gfCNCPoint3[1224] = {X 357.0844, Y 26.7729, Z -3.8333, A 0.000, B 0.000, C 0.000 }
gfCNCPoint3[1225] = {X 357.1951, Y 25.0733, Z -3.8333, A 0.000, B 0.000, C 0.000 }
gfCNCPoint3[1226] = {X 357.1435, Y 23.3709, Z -3.8333, A 0.000, B 0.000, C 0.000 }
gfCNCPoint3[1227] = {X 356.9299, Y 21.6811, Z -3.8333, A 0.000, B 0.000, C 0.000 }
gfCNCPoint3[1228] = {X 356.5958, Y 20.2415, Z -3.8333, A 0.000, B 0.000, C 0.000 }
gfCNCPoint3[1229] = {X 356.0861, Y 18.8543, Z -3.8333, A 0.000, B 0.000, C 0.000 }
gfCNCPoint3[1230] = {X 355.4086, Y 17.5409, Z -3.8333, A 0.000, B 0.000, C 0.000 }
gfCNCPoint3[1231] = {X 354.5737, Y 16.3214, Z -3.8333, A 0.000, B 0.000, C 0.000 }
gfCNCPoint3[1232] = {X 353.6956, Y 15.3423, Z -3.8333, A 0.000, B 0.000, C 0.000 }
gfCNCPoint3[1233] = {X 352.6863, Y 14.4990, Z -3.8333, A 0.000, B 0.000, C 0.000 }
gfCNCPoint3[1234] = {X 351.5666, Y 13.8090, Z -3.8333, A 0.000, B 0.000, C 0.000 }
gfCNCPoint3[1235] = {X 350.3596, Y 13.2864, Z -3.8333, A 0.000, B 0.000, C 0.000 }
gfCNCPoint3[1236] = {X 349.0902, Y 12.9422, Z -3.8333, A 0.000, B 0.000, C 0.000 }
gfCNCPoint3[1237] = {X 347.3476, Y 12.7251, Z -3.8333, A 0.000, B 0.000, C 0.000 }
gfCNCPoint3[1238] = {X 345.5915, Y 12.7393, Z -3.8333, A 0.000, B 0.000, C 0.000 }
gfCNCPoint3[1239] = {X 343.8527, Y 12.9848, Z -3.8333, A 0.000, B 0.000, C 0.000 }
gfCNCPoint3[1240] = {X 342.1613, Y 13.4572, Z -3.8333, A 0.000, B 0.000, C 0.000 }
gfCNCPoint3[1241] = {X 340.5469, Y 14.1483, Z -3.8333, A 0.000, B 0.000, C 0.000 }
gfCNCPoint3[1242] = {X 339.0376, Y 15.0460, Z -3.8333, A 0.000, B 0.000, C 0.000 }
gfCNCPoint3[1243] = {X 338.9896, Y 15.9040, Z -3.8333, A 0.000, B 0.000, C 0.000 }
gfCNCPoint3[1244] = {X 338.7758, Y 16.7364, Z -3.8333, A 0.000, B 0.000, C 0.000 }
gfCNCPoint3[1245] = {X 338.4043, Y 17.5112, Z -3.8333, A 0.000, B 0.000, C 0.000 }
gfCNCPoint3[1246] = {X 337.8893, Y 18.1991, Z -3.8333, A 0.000, B 0.000, C 0.000 }
gfCNCPoint3[1247] = {X 337.2504, Y 18.7738, Z -3.8333, A 0.000, B 0.000, C 0.000 }
gfCNCPoint3[1248] = {X 336.5606, Y 19.2813, Z -3.8333, A 0.000, B 0.000, C 0.000 }
gfCNCPoint3[1249] = {X 335.7284, Y 19.7495, Z -3.8333, A 0.000, B 0.000, C 0.000 }
gfCNCPoint3[1250] = {X 334.8148, Y 20.0271, Z -3.8333, A 0.000, B 0.000, C 0.000 }
gfCNCPoint3[1251] = {X 333.8628, Y 20.1012, Z -3.8333, A 0.000, B 0.000, C 0.000 }
gfCNCPoint3[1252] = {X 332.9173, Y 19.9681, Z -3.8333, A 0.000, B 0.000, C 0.000 }
gfCNCPoint3[1253] = {X 332.0228, Y 19.6341, Z -3.8333, A 0.000, B 0.000, C 0.000 }
gfCNCPoint3[1254] = {X 331.2213, Y 19.1151, Z -3.8333, A 0.000, B 0.000, C 0.000 }
gfCNCPoint3[1255] = {X 330.5507, Y 18.4353, Z -3.8333, A 0.000, B 0.000, C 0.000 }
gfCNCPoint3[1256] = {X 330.0425, Y 17.6269, Z -3.8333, A 0.000, B 0.000, C 0.000 }
gfCNCPoint3[1257] = {X 326.5223, Y 10.3852, Z -3.8333, A 0.000, B 0.000, C 0.000 }
gfCNCPoint3[1258] = {X 326.2154, Y 9.5469, Z -3.8333, A 0.000, B 0.000, C 0.000 }
gfCNCPoint3[1259] = {X 326.0841, Y 8.6639, Z -3.8333, A 0.000, B 0.000, C 0.000 }
gfCNCPoint3[1260] = {X 326.1338, Y 7.7725, Z -3.8333, A 0.000, B 0.000, C 0.000 }
gfCNCPoint3[1261] = {X 326.3623, Y 6.9096, Z -3.8333, A 0.000, B 0.000, C 0.000 }
gfCNCPoint3[1262] = {X 326.7603, Y 6.1105, Z -3.8333, A 0.000, B 0.000, C 0.000 }
gfCNCPoint3[1263] = {X 327.3114, Y 5.4082, Z -3.8333, A 0.000, B 0.000, C 0.000 }
gfCNCPoint3[1264] = {X 327.9929, Y 4.8316, Z -3.8333, A 0.000, B 0.000, C 0.000 }
gfCNCPoint3[1265] = {X 328.6647, Y 4.3715, Z -3.8333, A 0.000, B 0.000, C 0.000 }
gfCNCPoint3[1266] = {X 329.5525, Y 3.9111, Z -3.8333, A 0.000, B 0.000, C 0.000 }
gfCNCPoint3[1267] = {X 330.5213, Y 3.6631, Z -3.8333, A 0.000, B 0.000, C 0.000 }
gfCNCPoint3[1268] = {X 331.5211, Y 3.6402, Z -3.8333, A 0.000, B 0.000, C 0.000 }
gfCNCPoint3[1269] = {X 332.5003, Y 3.8437, Z -3.8333, A 0.000, B 0.000, C 0.000 }
gfCNCPoint3[1270] = {X 333.5103, Y 3.2689, Z -3.8333, A 0.000, B 0.000, C 0.000 }
gfCNCPoint3[1271] = {X 334.5430, Y 2.7360, Z -3.8333, A 0.000, B 0.000, C 0.000 }
gfCNCPoint3[1272] = {X 334.3316, Y 2.3050, Z -3.8333, A 0.000, B 0.000, C 0.000 }
gfCNCPoint3[1273] = {X 2.3035, Y 2.3050, Z -3.8333, A 0.000, B 0.000, C 0.000 }
gfCNCPoint3[1274] = {X 2.3035, Y 6.8597, Z -3.8333, A 0.000, B 0.000, C 0.000 }
gfCNCPoint3[1275] = {X 2.4041, Y 6.8798, Z -3.8333, A 0.000, B 0.000, C 0.000 }
gfCNCPoint3[1276] = {X 2.8649, Y 6.6913, Z -3.8333, A 0.000, B 0.000, C 0.000 }
gfCNCPoint3[1277] = {X 3.3320, Y 6.5189, Z -3.8333, A 0.000, B 0.000, C 0.000 }
gfCNCPoint3[1278] = {X 5.4373, Y 5.7870, Z -3.8333, A 0.000, B 0.000, C 0.000 }
gfCNCPoint3[1279] = {X 7.5978, Y 5.2386, Z -3.8333, A 0.000, B 0.000, C 0.000 }
gfCNCPoint3[1280] = {X 9.7973, Y 4.8776, Z -3.8333, A 0.000, B 0.000, C 0.000 }
gfCNCPoint3[1281] = {X 12.0197, Y 4.7069, Z -3.8333, A 0.000, B 0.000, C 0.000 }
gfCNCPoint3[1282] = {X 14.2486, Y 4.7276, Z -3.8333, A 0.000, B 0.000, C 0.000 }
gfCNCPoint3[1283] = {X 16.4674, Y 4.9396, Z -3.8333, A 0.000, B 0.000, C 0.000 }
gfCNCPoint3[1284] = {X 18.0965, Y 5.2204, Z -3.8333, A 0.000, B 0.000, C 0.000 }
gfCNCPoint3[1285] = {X 19.6967, Y 5.6352, Z -3.8333, A 0.000, B 0.000, C 0.000 }
gfCNCPoint3[1286] = {X 21.2571, Y 6.1811, Z -3.8333, A 0.000, B 0.000, C 0.000 }
gfCNCPoint3[1287] = {X 22.7668, Y 6.8545, Z -3.8333, A 0.000, B 0.000, C 0.000 }
gfCNCPoint3[1288] = {X 24.4883, Y 7.8186, Z -3.8333, A 0.000, B 0.000, C 0.000 }
gfCNCPoint3[1289] = {X 26.1061, Y 8.9481, Z -3.8333, A 0.000, B 0.000, C 0.000 }
gfCNCPoint3[1290] = {X 27.4003, Y 10.0783, Z -3.8333, A 0.000, B 0.000, C 0.000 }
gfCNCPoint3[1291] = {X 28.5612, Y 11.3450, Z -3.8333, A 0.000, B 0.000, C 0.000 }
gfCNCPoint3[1292] = {X 29.5745, Y 12.7325, Z -3.8333, A 0.000, B 0.000, C 0.000 }
gfCNCPoint3[1293] = {X 30.4278, Y 14.2239, Z -3.8333, A 0.000, B 0.000, C 0.000 }
gfCNCPoint3[1294] = {X 31.1104, Y 15.8006, Z -3.8333, A 0.000, B 0.000, C 0.000 }
gfCNCPoint3[1295] = {X 31.6697, Y 17.7362, Z -3.8333, A 0.000, B 0.000, C 0.000 }
gfCNCPoint3[1296] = {X 32.0027, Y 19.7232, Z -3.8333, A 0.000, B 0.000, C 0.000 }
gfCNCPoint3[1297] = {X 32.1050, Y 21.7354, Z -3.8333, A 0.000, B 0.000, C 0.000 }
gfCNCPoint3[1298] = {X 31.9753, Y 23.7459, Z -3.8333, A 0.000, B 0.000, C 0.000 }
gfCNCPoint3[1299] = {X 31.6152, Y 25.7282, Z -3.8333, A 0.000, B 0.000, C 0.000 }
gfCNCPoint3[1300] = {X 31.1690, Y 27.2346, Z -3.8333, A 0.000, B 0.000, C 0.000 }
gfCNCPoint3[1301] = {X 30.5588, Y 28.6823, Z -3.8333, A 0.000, B 0.000, C 0.000 }
gfCNCPoint3[1302] = {X 29.7921, Y 30.0536, Z -3.8333, A 0.000, B 0.000, C 0.000 }
gfCNCPoint3[1303] = {X 29.4475, Y 30.5712, Z -3.8333, A 0.000, B 0.000, C 0.000 }
gfCNCPoint3[1304] = {X 29.0806, Y 31.0733, Z -3.8333, A 0.000, B 0.000, C 0.000 }
gfCNCPoint3[1305] = {X 29.6385, Y 31.7919, Z -3.8333, A 0.000, B 0.000, C 0.000 }
gfCNCPoint3[1306] = {X 30.0955, Y 32.5786, Z -3.8333, A 0.000, B 0.000, C 0.000 }
gfCNCPoint3[1307] = {X 33.1423, Y 38.8726, Z -3.8333, A 0.000, B 0.000, C 0.000 }
gfCNCPoint3[1308] = {X 33.5391, Y 39.8957, Z -3.8333, A 0.000, B 0.000, C 0.000 }
gfCNCPoint3[1309] = {X 33.7662, Y 40.9694, Z -3.8333, A 0.000, B 0.000, C 0.000 }
gfCNCPoint3[1310] = {X 33.8177, Y 42.0656, Z -3.8333, A 0.000, B 0.000, C 0.000 }
gfCNCPoint3[1311] = {X 33.7164, Y 43.0266, Z -3.8333, A 0.000, B 0.000, C 0.000 }
gfCNCPoint3[1312] = {X 33.4799, Y 43.9636, Z -3.8333, A 0.000, B 0.000, C 0.000 }
gfCNCPoint3[1313] = {X 33.1103, Y 44.8630, Z -3.8333, A 0.000, B 0.000, C 0.000 }
gfCNCPoint3[1314] = {X 32.6161, Y 45.7005, Z -3.8333, A 0.000, B 0.000, C 0.000 }
gfCNCPoint3[1315] = {X 32.0075, Y 46.4590, Z -3.8333, A 0.000, B 0.000, C 0.000 }
gfCNCPoint3[1316] = {X 31.2970, Y 47.1229, Z -3.8333, A 0.000, B 0.000, C 0.000 }
gfCNCPoint3[1317] = {X 30.7593, Y 47.5577, Z -3.8333, A 0.000, B 0.000, C 0.000 }
gfCNCPoint3[1318] = {X 29.8533, Y 48.1757, Z -3.8333, A 0.000, B 0.000, C 0.000 }
gfCNCPoint3[1319] = {X 28.8600, Y 48.6403, Z -3.8333, A 0.000, B 0.000, C 0.000 }
gfCNCPoint3[1320] = {X 27.8050, Y 48.9396, Z -3.8333, A 0.000, B 0.000, C 0.000 }
gfCNCPoint3[1321] = {X 26.7156, Y 49.0659, Z -3.8333, A 0.000, B 0.000, C 0.000 }
gfCNCPoint3[1322] = {X 25.6202, Y 49.0158, Z -3.8333, A 0.000, B 0.000, C 0.000 }
gfCNCPoint3[1323] = {X 23.9315, Y 49.8548, Z -3.8333, A 0.000, B 0.000, C 0.000 }
gfCNCPoint3[1324] = {X 22.1957, Y 50.5913, Z -3.8333, A 0.000, B 0.000, C 0.000 }
gfCNCPoint3[1325] = {X 20.4190, Y 51.2227, Z -3.8333, A 0.000, B 0.000, C 0.000 }
gfCNCPoint3[1326] = {X 18.3991, Y 51.7971, Z -3.8333, A 0.000, B 0.000, C 0.000 }
gfCNCPoint3[1327] = {X 16.3386, Y 52.2022, Z -3.8333, A 0.000, B 0.000, C 0.000 }
gfCNCPoint3[1328] = {X 14.2517, Y 52.4352, Z -3.8333, A 0.000, B 0.000, C 0.000 }
gfCNCPoint3[1329] = {X 12.1526, Y 52.4947, Z -3.8333, A 0.000, B 0.000, C 0.000 }
gfCNCPoint3[1330] = {X 10.0558, Y 52.3800, Z -3.8333, A 0.000, B 0.000, C 0.000 }
gfCNCPoint3[1331] = {X 7.9757, Y 52.0921, Z -3.8333, A 0.000, B 0.000, C 0.000 }
gfCNCPoint3[1332] = {X 6.6905, Y 51.8245, Z -3.8333, A 0.000, B 0.000, C 0.000 }
gfCNCPoint3[1333] = {X 5.4261, Y 51.4714, Z -3.8333, A 0.000, B 0.000, C 0.000 }
gfCNCPoint3[1334] = {X 3.8369, Y 50.8930, Z -3.8333, A 0.000, B 0.000, C 0.000 }
gfCNCPoint3[1335] = {X 2.3035, Y 50.1795, Z -3.8333, A 0.000, B 0.000, C 0.000 }
gfCNCPoint3[1336] = {X 2.3035, Y 97.6950, Z -3.8333, A 0.000, B 0.000, C 0.000 }
gfCNCPoint3[1337] = {X 120.1200, Y 97.6950, Z -3.8333, A 0.000, B 0.000, C 0.000 }
gfCNCPoint3[1338] = {X 120.1200, Y 97.0659, Z -3.8333, A 0.000, B 0.000, C 0.000 }
gfCNCPoint3[1339] = {X 120.2339, Y 96.0179, Z -3.8333, A 0.000, B 0.000, C 0.000 }
gfCNCPoint3[1340] = {X 120.5702, Y 95.0187, Z -3.8333, A 0.000, B 0.000, C 0.000 }
gfCNCPoint3[1341] = {X 121.1132, Y 94.1151, Z -3.8333, A 0.000, B 0.000, C 0.000 }
gfCNCPoint3[1342] = {X 121.8376, Y 93.3492, Z -3.8333, A 0.000, B 0.000, C 0.000 }
gfCNCPoint3[1343] = {X 122.7096, Y 92.7568, Z -3.8333, A 0.000, B 0.000, C 0.000 }
gfCNCPoint3[1344] = {X 123.6885, Y 92.3655, Z -3.8333, A 0.000, B 0.000, C 0.000 }
gfCNCPoint3[1345] = {X 124.7286, Y 92.1935, Z -3.8333, A 0.000, B 0.000, C 0.000 }
gfCNCPoint3[1346] = {X 124.7867, Y 92.1787, Z -3.8333, A 0.000, B 0.000, C 0.000 }
gfCNCPoint3[1347] = {X 124.8457, Y 92.1679, Z -3.8333, A 0.000, B 0.000, C 0.000 }
gfCNCPoint3[1348] = {X 125.3649, Y 92.0908, Z -3.8333, A 0.000, B 0.000, C 0.000 }
gfCNCPoint3[1349] = {X 126.0998, Y 91.9697, Z -3.8333, A 0.000, B 0.000, C 0.000 }
gfCNCPoint3[1350] = {X 126.8256, Y 91.8023, Z -3.8333, A 0.000, B 0.000, C 0.000 }
gfCNCPoint3[1351] = {X 127.9736, Y 90.7130, Z -3.8333, A 0.000, B 0.000, C 0.000 }
gfCNCPoint3[1352] = {X 129.0632, Y 89.5654, Z -3.8333, A 0.000, B 0.000, C 0.000 }
gfCNCPoint3[1353] = {X 154.9462, Y 61.1423, Z -3.8333, A 0.000, B 0.000, C 0.000 }
gfCNCPoint3[1354] = {X 154.6593, Y 60.4497, Z -3.8333, A 0.000, B 0.000, C 0.000 }
gfCNCPoint3[1355] = {X 154.4819, Y 59.7213, Z -3.8333, A 0.000, B 0.000, C 0.000 }
gfCNCPoint3[1356] = {X 154.4181, Y 58.9744, Z -3.8333, A 0.000, B 0.000, C 0.000 }
gfCNCPoint3[1357] = {X 154.4180, Y 58.0000, Z -3.8333, A 0.000, B 0.000, C 0.000 }
gfCNCPoint3[1358] = {X 154.5117, Y 57.0480, Z -3.8333, A 0.000, B 0.000, C 0.000 }
gfCNCPoint3[1359] = {X 154.7894, Y 56.1325, Z -3.8333, A 0.000, B 0.000, C 0.000 }
gfCNCPoint3[1360] = {X 155.2404, Y 55.2888, Z -3.8333, A 0.000, B 0.000, C 0.000 }
gfCNCPoint3[1361] = {X 155.8473, Y 54.5493, Z -3.8333, A 0.000, B 0.000, C 0.000 }
gfCNCPoint3[1362] = {X 156.5868, Y 53.9424, Z -3.8333, A 0.000, B 0.000, C 0.000 }
gfCNCPoint3[1363] = {X 157.4305, Y 53.4915, Z -3.8333, A 0.000, B 0.000, C 0.000 }
gfCNCPoint3[1364] = {X 158.3459, Y 53.2138, Z -3.8333, A 0.000, B 0.000, C 0.000 }
gfCNCPoint3[1365] = {X 159.2980, Y 53.1200, Z -3.8333, A 0.000, B 0.000, C 0.000 }
gfCNCPoint3[1366] = {X 178.5335, Y 53.1200, Z -3.8333, A 0.000, B 0.000, C 0.000 }
gfCNCPoint3[1367] = {X 179.4855, Y 53.2138, Z -3.8333, A 0.000, B 0.000, C 0.000 }
gfCNCPoint3[1368] = {X 180.4010, Y 53.4915, Z -3.8333, A 0.000, B 0.000, C 0.000 }
gfCNCPoint3[1369] = {X 181.2447, Y 53.9424, Z -3.8333, A 0.000, B 0.000, C 0.000 }
gfCNCPoint3[1370] = {X 181.9842, Y 54.5493, Z -3.8333, A 0.000, B 0.000, C 0.000 }
gfCNCPoint3[1371] = {X 182.5911, Y 55.2888, Z -3.8333, A 0.000, B 0.000, C 0.000 }
gfCNCPoint3[1372] = {X 183.0420, Y 56.1325, Z -3.8333, A 0.000, B 0.000, C 0.000 }
gfCNCPoint3[1373] = {X 183.3197, Y 57.0480, Z -3.8333, A 0.000, B 0.000, C 0.000 }
gfCNCPoint3[1374] = {X 183.4135, Y 58.0000, Z -3.8333, A 0.000, B 0.000, C 0.000 }
gfCNCPoint3[1375] = {X 183.4133, Y 58.9744, Z -3.8333, A 0.000, B 0.000, C 0.000 }
gfCNCPoint3[1376] = {X 183.3512, Y 59.7113, Z -3.8333, A 0.000, B 0.000, C 0.000 }
gfCNCPoint3[1377] = {X 183.1784, Y 60.4304, Z -3.8333, A 0.000, B 0.000, C 0.000 }
gfCNCPoint3[1378] = {X 182.8990, Y 61.1152, Z -3.8333, A 0.000, B 0.000, C 0.000 }
gfCNCPoint3[1379] = {X 209.8913, Y 90.5758, Z -3.8333, A 0.000, B 0.000, C 0.000 }
gfCNCPoint3[1380] = {X 210.5201, Y 91.2137, Z -3.8333, A 0.000, B 0.000, C 0.000 }
gfCNCPoint3[1381] = {X 211.1937, Y 91.8042, Z -3.8333, A 0.000, B 0.000, C 0.000 }
gfCNCPoint3[1382] = {X 211.3597, Y 91.9086, Z -3.8333, A 0.000, B 0.000, C 0.000 }
gfCNCPoint3[1383] = {X 211.5461, Y 91.9696, Z -3.8333, A 0.000, B 0.000, C 0.000 }
gfCNCPoint3[1384] = {X 212.2018, Y 92.1098, Z -3.8333, A 0.000, B 0.000, C 0.000 }
gfCNCPoint3[1385] = {X 213.4083, Y 92.2618, Z -3.8333, A 0.000, B 0.000, C 0.000 }
gfCNCPoint3[1386] = {X 214.4425, Y 92.1756, Z -3.8333, A 0.000, B 0.000, C 0.000 }
gfCNCPoint3[1387] = {X 215.4785, Y 92.1166, Z -3.8333, A 0.000, B 0.000, C 0.000 }
gfCNCPoint3[1388] = {X 216.0525, Y 92.0568, Z -3.8333, A 0.000, B 0.000, C 0.000 }
gfCNCPoint3[1389] = {X 216.6054, Y 91.8915, Z -3.8333, A 0.000, B 0.000, C 0.000 }
gfCNCPoint3[1390] = {X 217.1180, Y 91.6265, Z -3.8333, A 0.000, B 0.000, C 0.000 }
gfCNCPoint3[1391] = {X 244.6013, Y 74.0195, Z -3.8333, A 0.000, B 0.000, C 0.000 }
gfCNCPoint3[1392] = {X 221.4278, Y 64.9254, Z -3.8333, A 0.000, B 0.000, C 0.000 }
gfCNCPoint3[1393] = {X 219.7200, Y 64.3531, Z -3.8333, A 0.000, B 0.000, C 0.000 }
gfCNCPoint3[1394] = {X 217.9579, Y 63.9800, Z -3.8333, A 0.000, B 0.000, C 0.000 }
gfCNCPoint3[1395] = {X 216.1647, Y 63.8112, Z -3.8333, A 0.000, B 0.000, C 0.000 }
gfCNCPoint3[1396] = {X 215.1121, Y 63.6594, Z -3.8333, A 0.000, B 0.000, C 0.000 }
gfCNCPoint3[1397] = {X 214.1174, Y 63.2832, Z -3.8333, A 0.000, B 0.000, C 0.000 }
gfCNCPoint3[1398] = {X 213.2278, Y 62.7005, Z -3.8333, A 0.000, B 0.000, C 0.000 }
gfCNCPoint3[1399] = {X 212.4856, Y 61.9389, Z -3.8333, A 0.000, B 0.000, C 0.000 }
gfCNCPoint3[1400] = {X 211.9260, Y 61.0346, Z -3.8333, A 0.000, B 0.000, C 0.000 }
gfCNCPoint3[1401] = {X 211.5756, Y 60.0305, Z -3.8333, A 0.000, B 0.000, C 0.000 }
gfCNCPoint3[1402] = {X 211.4510, Y 58.9744, Z -3.8333, A 0.000, B 0.000, C 0.000 }
gfCNCPoint3[1403] = {X 211.4508, Y 58.0000, Z -3.8333, A 0.000, B 0.000, C 0.000 }
gfCNCPoint3[1404] = {X 211.5446, Y 57.0480, Z -3.8333, A 0.000, B 0.000, C 0.000 }
gfCNCPoint3[1405] = {X 211.8223, Y 56.1325, Z -3.8333, A 0.000, B 0.000, C 0.000 }
gfCNCPoint3[1406] = {X 212.2732, Y 55.2888, Z -3.8333, A 0.000, B 0.000, C 0.000 }
gfCNCPoint3[1407] = {X 212.8801, Y 54.5493, Z -3.8333, A 0.000, B 0.000, C 0.000 }
gfCNCPoint3[1408] = {X 213.6196, Y 53.9424, Z -3.8333, A 0.000, B 0.000, C 0.000 }
gfCNCPoint3[1409] = {X 214.4633, Y 53.4915, Z -3.8333, A 0.000, B 0.000, C 0.000 }
gfCNCPoint3[1410] = {X 215.3788, Y 53.2138, Z -3.8333, A 0.000, B 0.000, C 0.000 }
gfCNCPoint3[1411] = {X 216.3308, Y 53.1200, Z -3.8333, A 0.000, B 0.000, C 0.000 }
gfCNCPoint3[1412] = {X 237.2617, Y 53.1200, Z -3.8333, A 0.000, B 0.000, C 0.000 }
gfCNCPoint3[1413] = {X 238.3265, Y 53.2376, Z -3.8333, A 0.000, B 0.000, C 0.000 }
gfCNCPoint3[1414] = {X 239.3400, Y 53.5847, Z -3.8333, A 0.000, B 0.000, C 0.000 }
gfCNCPoint3[1415] = {X 240.2534, Y 54.1446, Z -3.8333, A 0.000, B 0.000, C 0.000 }
gfCNCPoint3[1416] = {X 241.0226, Y 54.8903, Z -3.8333, A 0.000, B 0.000, C 0.000 }
gfCNCPoint3[1417] = {X 241.6105, Y 55.7859, Z -3.8333, A 0.000, B 0.000, C 0.000 }
gfCNCPoint3[1418] = {X 241.9888, Y 56.7881, Z -3.8333, A 0.000, B 0.000, C 0.000 }
gfCNCPoint3[1419] = {X 242.1393, Y 57.8488, Z -3.8333, A 0.000, B 0.000, C 0.000 }
gfCNCPoint3[1420] = {X 247.6958, Y 60.0148, Z -3.8333, A 0.000, B 0.000, C 0.000 }
gfCNCPoint3[1421] = {X 275.0731, Y 70.8777, Z -3.8333, A 0.000, B 0.000, C 0.000 }
gfCNCPoint3[1422] = {X 275.0726, Y 63.6742, Z -3.8333, A 0.000, B 0.000, C 0.000 }
gfCNCPoint3[1423] = {X 274.0643, Y 63.3058, Z -3.8333, A 0.000, B 0.000, C 0.000 }
gfCNCPoint3[1424] = {X 273.1609, Y 62.7260, Z -3.8333, A 0.000, B 0.000, C 0.000 }
gfCNCPoint3[1425] = {X 272.4062, Y 61.9626, Z -3.8333, A 0.000, B 0.000, C 0.000 }
gfCNCPoint3[1426] = {X 271.8366, Y 61.0527, Z -3.8333, A 0.000, B 0.000, C 0.000 }
gfCNCPoint3[1427] = {X 271.4797, Y 60.0403, Z -3.8333, A 0.000, B 0.000, C 0.000 }
gfCNCPoint3[1428] = {X 271.3529, Y 58.9744, Z -3.8333, A 0.000, B 0.000, C 0.000 }
gfCNCPoint3[1429] = {X 271.3527, Y 58.0000, Z -3.8333, A 0.000, B 0.000, C 0.000 }
gfCNCPoint3[1430] = {X 271.4465, Y 57.0480, Z -3.8333, A 0.000, B 0.000, C 0.000 }
gfCNCPoint3[1431] = {X 271.7242, Y 56.1325, Z -3.8333, A 0.000, B 0.000, C 0.000 }
gfCNCPoint3[1432] = {X 272.1751, Y 55.2888, Z -3.8333, A 0.000, B 0.000, C 0.000 }
gfCNCPoint3[1433] = {X 272.7820, Y 54.5493, Z -3.8333, A 0.000, B 0.000, C 0.000 }
gfCNCPoint3[1434] = {X 273.5215, Y 53.9424, Z -3.8333, A 0.000, B 0.000, C 0.000 }
gfCNCPoint3[1435] = {X 274.3652, Y 53.4915, Z -3.8333, A 0.000, B 0.000, C 0.000 }
gfCNCPoint3[1436] = {X 275.2806, Y 53.2138, Z -3.8333, A 0.000, B 0.000, C 0.000 }
gfCNCPoint3[1437] = {X 276.2327, Y 53.1200, Z -3.8333, A 0.000, B 0.000, C 0.000 }
gfCNCPoint3[1438] = {X 292.7731, Y 53.1200, Z -3.8333, A 0.000, B 0.000, C 0.000 }
gfCNCPoint3[1439] = {X 293.7251, Y 53.2138, Z -3.8333, A 0.000, B 0.000, C 0.000 }
gfCNCPoint3[1440] = {X 294.6406, Y 53.4915, Z -3.8333, A 0.000, B 0.000, C 0.000 }
gfCNCPoint3[1441] = {X 295.4843, Y 53.9424, Z -3.8333, A 0.000, B 0.000, C 0.000 }
gfCNCPoint3[1442] = {X 296.2238, Y 54.5493, Z -3.8333, A 0.000, B 0.000, C 0.000 }
gfCNCPoint3[1443] = {X 296.8307, Y 55.2888, Z -3.8333, A 0.000, B 0.000, C 0.000 }
gfCNCPoint3[1444] = {X 297.2816, Y 56.1325, Z -3.8333, A 0.000, B 0.000, C 0.000 }
gfCNCPoint3[1445] = {X 297.5593, Y 57.0480, Z -3.8333, A 0.000, B 0.000, C 0.000 }
gfCNCPoint3[1446] = {X 297.6531, Y 58.0000, Z -3.8333, A 0.000, B 0.000, C 0.000 }
gfCNCPoint3[1447] = {X 297.6531, Y 58.9370, Z -3.8333, A 0.000, B 0.000, C 0.000 }
gfCNCPoint3[1448] = {X 297.5307, Y 60.0092, Z -3.8333, A 0.000, B 0.000, C 0.000 }
gfCNCPoint3[1449] = {X 297.1764, Y 61.0286, Z -3.8333, A 0.000, B 0.000, C 0.000 }
gfCNCPoint3[1450] = {X 296.6074, Y 61.9456, Z -3.8333, A 0.000, B 0.000, C 0.000 }
gfCNCPoint3[1451] = {X 295.8514, Y 62.7156, Z -3.8333, A 0.000, B 0.000, C 0.000 }
gfCNCPoint3[1452] = {X 294.9451, Y 63.3014, Z -3.8333, A 0.000, B 0.000, C 0.000 }
gfCNCPoint3[1453] = {X 293.9324, Y 63.6745, Z -3.8333, A 0.000, B 0.000, C 0.000 }
gfCNCPoint3[1454] = {X 293.9324, Y 92.3204, Z -3.8333, A 0.000, B 0.000, C 0.000 }
gfCNCPoint3[1455] = {X 294.9449, Y 92.6960, Z -3.8333, A 0.000, B 0.000, C 0.000 }
gfCNCPoint3[1456] = {X 295.8509, Y 93.2837, Z -3.8333, A 0.000, B 0.000, C 0.000 }
gfCNCPoint3[1457] = {X 296.6066, Y 94.0552, Z -3.8333, A 0.000, B 0.000, C 0.000 }
gfCNCPoint3[1458] = {X 297.1754, Y 94.9731, Z -3.8333, A 0.000, B 0.000, C 0.000 }
gfCNCPoint3[1459] = {X 297.5300, Y 95.9932, Z -3.8333, A 0.000, B 0.000, C 0.000 }
gfCNCPoint3[1460] = {X 297.6531, Y 97.0661, Z -3.8333, A 0.000, B 0.000, C 0.000 }
gfCNCPoint3[1461] = {X 297.6531, Y 97.6950, Z -3.8333, A 0.000, B 0.000, C 0.000 }
gfCNCPoint3[1462] = {X 297.1731, Y 97.6950, Z -3.8333, A 0.000, B 0.000, C 0.000 }
gfCNCPoint3[1463] = {X 297.1731, Y 98.0000, Z -3.8333, A 0.000, B 0.000, C 0.000 }
gfCNCPoint3[1464] = {X 297.0628, Y 98.9791, Z -3.8333, A 0.000, B 0.000, C 0.000 }
gfCNCPoint3[1465] = {X 296.7373, Y 99.9091, Z -3.8333, A 0.000, B 0.000, C 0.000 }
gfCNCPoint3[1466] = {X 296.2131, Y 100.7434, Z -3.8333, A 0.000, B 0.000, C 0.000 }
gfCNCPoint3[1467] = {X 295.5164, Y 101.4401, Z -3.8333, A 0.000, B 0.000, C 0.000 }
gfCNCPoint3[1468] = {X 294.6822, Y 101.9643, Z -3.8333, A 0.000, B 0.000, C 0.000 }
gfCNCPoint3[1469] = {X 293.7522, Y 102.2897, Z -3.8333, A 0.000, B 0.000, C 0.000 }
gfCNCPoint3[1470] = {X 292.7731, Y 102.4000, Z -3.8333, A 0.000, B 0.000, C 0.000 }
gfCNCPoint3[1471] = {X 276.2327, Y 102.4000, Z -3.8333, A 0.000, B 0.000, C 0.000 }
gfCNCPoint3[1472] = {X 275.2536, Y 102.2897, Z -3.8333, A 0.000, B 0.000, C 0.000 }
gfCNCPoint3[1473] = {X 274.3236, Y 101.9643, Z -3.8333, A 0.000, B 0.000, C 0.000 }
gfCNCPoint3[1474] = {X 273.4893, Y 101.4401, Z -3.8333, A 0.000, B 0.000, C 0.000 }
gfCNCPoint3[1475] = {X 272.7926, Y 100.7434, Z -3.8333, A 0.000, B 0.000, C 0.000 }
gfCNCPoint3[1476] = {X 272.2684, Y 99.9091, Z -3.8333, A 0.000, B 0.000, C 0.000 }
gfCNCPoint3[1477] = {X 271.9430, Y 98.9791, Z -3.8333, A 0.000, B 0.000, C 0.000 }
gfCNCPoint3[1478] = {X 271.8327, Y 98.0000, Z -3.8333, A 0.000, B 0.000, C 0.000 }
gfCNCPoint3[1479] = {X 271.8329, Y 97.0190, Z -3.8333, A 0.000, B 0.000, C 0.000 }
gfCNCPoint3[1480] = {X 271.9305, Y 96.1432, Z -3.8333, A 0.000, B 0.000, C 0.000 }
gfCNCPoint3[1481] = {X 272.2006, Y 95.3045, Z -3.8333, A 0.000, B 0.000, C 0.000 }
gfCNCPoint3[1482] = {X 272.6325, Y 94.5364, Z -3.8333, A 0.000, B 0.000, C 0.000 }
gfCNCPoint3[1483] = {X 273.2087, Y 93.8698, Z -3.8333, A 0.000, B 0.000, C 0.000 }
gfCNCPoint3[1484] = {X 273.9062, Y 93.3313, Z -3.8333, A 0.000, B 0.000, C 0.000 }
gfCNCPoint3[1485] = {X 274.6970, Y 92.9426, Z -3.8333, A 0.000, B 0.000, C 0.000 }
gfCNCPoint3[1486] = {X 275.5494, Y 92.7193, Z -3.8333, A 0.000, B 0.000, C 0.000 }
gfCNCPoint3[1487] = {X 275.5494, Y 85.6495, Z -3.8333, A 0.000, B 0.000, C 0.000 }
gfCNCPoint3[1488] = {X 262.6481, Y 80.5922, Z -3.8333, A 0.000, B 0.000, C 0.000 }
gfCNCPoint3[1489] = {X 262.3197, Y 80.7991, Z -3.8333, A 0.000, B 0.000, C 0.000 }
gfCNCPoint3[1490] = {X 237.8767, Y 96.6314, Z -3.8333, A 0.000, B 0.000, C 0.000 }
gfCNCPoint3[1491] = {X 237.8798, Y 97.0659, Z -3.8333, A 0.000, B 0.000, C 0.000 }
gfCNCPoint3[1492] = {X 237.8798, Y 98.0000, Z -3.8333, A 0.000, B 0.000, C 0.000 }
gfCNCPoint3[1493] = {X 237.7695, Y 98.9791, Z -3.8333, A 0.000, B 0.000, C 0.000 }
gfCNCPoint3[1494] = {X 237.4440, Y 99.9091, Z -3.8333, A 0.000, B 0.000, C 0.000 }
gfCNCPoint3[1495] = {X 236.9198, Y 100.7434, Z -3.8333, A 0.000, B 0.000, C 0.000 }
gfCNCPoint3[1496] = {X 236.2231, Y 101.4401, Z -3.8333, A 0.000, B 0.000, C 0.000 }
gfCNCPoint3[1497] = {X 235.3889, Y 101.9643, Z -3.8333, A 0.000, B 0.000, C 0.000 }
gfCNCPoint3[1498] = {X 234.4589, Y 102.2897, Z -3.8333, A 0.000, B 0.000, C 0.000 }
gfCNCPoint3[1499] = {X 233.4798, Y 102.4000, Z -3.8333, A 0.000, B 0.000, C 0.000 }
gfCNCPoint3[1500] = {X 214.1790, Y 102.4000, Z -3.8333, A 0.000, B 0.000, C 0.000 }
gfCNCPoint3[1501] = {X 213.7862, Y 102.3824, Z -3.8333, A 0.000, B 0.000, C 0.000 }
gfCNCPoint3[1502] = {X 213.3966, Y 102.3299, Z -3.8333, A 0.000, B 0.000, C 0.000 }
gfCNCPoint3[1503] = {X 213.0069, Y 102.3824, Z -3.8333, A 0.000, B 0.000, C 0.000 }
gfCNCPoint3[1504] = {X 212.6141, Y 102.4000, Z -3.8333, A 0.000, B 0.000, C 0.000 }
gfCNCPoint3[1505] = {X 194.9870, Y 102.4000, Z -3.8333, A 0.000, B 0.000, C 0.000 }
gfCNCPoint3[1506] = {X 194.0079, Y 102.2897, Z -3.8333, A 0.000, B 0.000, C 0.000 }
gfCNCPoint3[1507] = {X 193.0779, Y 101.9643, Z -3.8333, A 0.000, B 0.000, C 0.000 }
gfCNCPoint3[1508] = {X 192.2436, Y 101.4401, Z -3.8333, A 0.000, B 0.000, C 0.000 }
gfCNCPoint3[1509] = {X 191.5469, Y 100.7434, Z -3.8333, A 0.000, B 0.000, C 0.000 }
gfCNCPoint3[1510] = {X 191.0227, Y 99.9091, Z -3.8333, A 0.000, B 0.000, C 0.000 }
gfCNCPoint3[1511] = {X 190.6973, Y 98.9791, Z -3.8333, A 0.000, B 0.000, C 0.000 }
gfCNCPoint3[1512] = {X 190.5870, Y 98.0000, Z -3.8333, A 0.000, B 0.000, C 0.000 }
gfCNCPoint3[1513] = {X 190.5870, Y 97.0659, Z -3.8333, A 0.000, B 0.000, C 0.000 }
gfCNCPoint3[1514] = {X 190.6897, Y 96.1207, Z -3.8333, A 0.000, B 0.000, C 0.000 }
gfCNCPoint3[1515] = {X 190.9931, Y 95.2196, Z -3.8333, A 0.000, B 0.000, C 0.000 }
gfCNCPoint3[1516] = {X 191.4830, Y 94.4047, Z -3.8333, A 0.000, B 0.000, C 0.000 }
gfCNCPoint3[1517] = {X 188.5295, Y 91.1802, Z -3.8333, A 0.000, B 0.000, C 0.000 }
gfCNCPoint3[1518] = {X 150.1254, Y 91.1802, Z -3.8333, A 0.000, B 0.000, C 0.000 }
gfCNCPoint3[1519] = {X 147.2494, Y 94.3664, Z -3.8333, A 0.000, B 0.000, C 0.000 }
gfCNCPoint3[1520] = {X 147.7554, Y 95.1907, Z -3.8333, A 0.000, B 0.000, C 0.000 }
gfCNCPoint3[1521] = {X 148.0703, Y 96.1051, Z -3.8333, A 0.000, B 0.000, C 0.000 }
gfCNCPoint3[1522] = {X 148.1791, Y 97.0661, Z -3.8333, A 0.000, B 0.000, C 0.000 }
gfCNCPoint3[1523] = {X 148.1791, Y 98.0000, Z -3.8333, A 0.000, B 0.000, C 0.000 }
gfCNCPoint3[1524] = {X 148.0688, Y 98.9791, Z -3.8333, A 0.000, B 0.000, C 0.000 }
gfCNCPoint3[1525] = {X 147.7434, Y 99.9091, Z -3.8333, A 0.000, B 0.000, C 0.000 }
gfCNCPoint3[1526] = {X 147.2192, Y 100.7434, Z -3.8333, A 0.000, B 0.000, C 0.000 }
gfCNCPoint3[1527] = {X 146.5225, Y 101.4401, Z -3.8333, A 0.000, B 0.000, C 0.000 }
gfCNCPoint3[1528] = {X 145.6882, Y 101.9643, Z -3.8333, A 0.000, B 0.000, C 0.000 }
gfCNCPoint3[1529] = {X 144.7582, Y 102.2897, Z -3.8333, A 0.000, B 0.000, C 0.000 }
gfCNCPoint3[1530] = {X 143.7791, Y 102.4000, Z -3.8333, A 0.000, B 0.000, C 0.000 }
gfCNCPoint3[1531] = {X 125.0000, Y 102.4000, Z -3.8333, A 0.000, B 0.000, C 0.000 }
gfCNCPoint3[1532] = {X 124.0209, Y 102.2897, Z -3.8333, A 0.000, B 0.000, C 0.000 }
gfCNCPoint3[1533] = {X 123.0909, Y 101.9643, Z -3.8333, A 0.000, B 0.000, C 0.000 }
gfCNCPoint3[1534] = {X 122.2566, Y 101.4401, Z -3.8333, A 0.000, B 0.000, C 0.000 }
gfCNCPoint3[1535] = {X 121.5599, Y 100.7434, Z -3.8333, A 0.000, B 0.000, C 0.000 }
gfCNCPoint3[1536] = {X 121.0357, Y 99.9091, Z -3.8333, A 0.000, B 0.000, C 0.000 }
gfCNCPoint3[1537] = {X 120.7103, Y 98.9791, Z -3.8333, A 0.000, B 0.000, C 0.000 }
gfCNCPoint3[1538] = {X 120.6000, Y 98.0000, Z -3.8333, A 0.000, B 0.000, C 0.000 }
gfCNCPoint3[1539] = {X 120.6000, Y 97.0659, Z -3.8333, A 0.000, B 0.000, C 0.000 }
gfCNCPoint3[1540] = {X 120.7047, Y 96.1120, Z -3.8333, A 0.000, B 0.000, C 0.000 }
gfCNCPoint3[1541] = {X 121.0137, Y 95.2034, Z -3.8333, A 0.000, B 0.000, C 0.000 }
gfCNCPoint3[1542] = {X 121.5123, Y 94.3834, Z -3.8333, A 0.000, B 0.000, C 0.000 }
gfCNCPoint3[1543] = {X 122.1769, Y 93.6910, Z -3.8333, A 0.000, B 0.000, C 0.000 }
gfCNCPoint3[1544] = {X 122.9757, Y 93.1592, Z -3.8333, A 0.000, B 0.000, C 0.000 }
gfCNCPoint3[1545] = {X 123.8709, Y 92.8133, Z -3.8333, A 0.000, B 0.000, C 0.000 }
gfCNCPoint3[1546] = {X 124.8198, Y 92.6696, Z -3.8333, A 0.000, B 0.000, C 0.000 }
gfCNCPoint3[1547] = {X 124.8671, Y 92.6531, Z -3.8333, A 0.000, B 0.000, C 0.000 }
gfCNCPoint3[1548] = {X 124.9162, Y 92.6427, Z -3.8333, A 0.000, B 0.000, C 0.000 }
gfCNCPoint3[1549] = {X 125.4412, Y 92.5648, Z -3.8333, A 0.000, B 0.000, C 0.000 }
gfCNCPoint3[1550] = {X 126.2566, Y 92.4278, Z -3.8333, A 0.000, B 0.000, C 0.000 }
gfCNCPoint3[1551] = {X 127.0610, Y 92.2360, Z -3.8333, A 0.000, B 0.000, C 0.000 }
gfCNCPoint3[1552] = {X 128.2728, Y 91.0926, Z -3.8333, A 0.000, B 0.000, C 0.000 }
gfCNCPoint3[1553] = {X 129.4210, Y 89.8854, Z -3.8333, A 0.000, B 0.000, C 0.000 }
gfCNCPoint3[1554] = {X 133.5081, Y 85.3895, Z -3.8333, A 0.000, B 0.000, C 0.000 }
gfCNCPoint3[1555] = {X 155.5329, Y 61.2109, Z -3.8333, A 0.000, B 0.000, C 0.000 }
gfCNCPoint3[1556] = {X 155.1840, Y 60.4948, Z -3.8333, A 0.000, B 0.000, C 0.000 }
gfCNCPoint3[1557] = {X 154.9701, Y 59.7274, Z -3.8333, A 0.000, B 0.000, C 0.000 }
gfCNCPoint3[1558] = {X 154.8980, Y 58.9340, Z -3.8333, A 0.000, B 0.000, C 0.000 }
gfCNCPoint3[1559] = {X 154.8980, Y 58.0000, Z -3.8333, A 0.000, B 0.000, C 0.000 }
gfCNCPoint3[1560] = {X 155.0083, Y 57.0209, Z -3.8333, A 0.000, B 0.000, C 0.000 }
gfCNCPoint3[1561] = {X 155.3337, Y 56.0909, Z -3.8333, A 0.000, B 0.000, C 0.000 }
gfCNCPoint3[1562] = {X 155.8579, Y 55.2566, Z -3.8333, A 0.000, B 0.000, C 0.000 }
gfCNCPoint3[1563] = {X 156.5546, Y 54.5599, Z -3.8333, A 0.000, B 0.000, C 0.000 }
gfCNCPoint3[1564] = {X 157.3889, Y 54.0357, Z -3.8333, A 0.000, B 0.000, C 0.000 }
gfCNCPoint3[1565] = {X 158.3189, Y 53.7103, Z -3.8333, A 0.000, B 0.000, C 0.000 }
gfCNCPoint3[1566] = {X 159.2980, Y 53.6000, Z -3.8333, A 0.000, B 0.000, C 0.000 }
gfCNCPoint3[1567] = {X 178.5335, Y 53.6000, Z -3.8333, A 0.000, B 0.000, C 0.000 }
gfCNCPoint3[1568] = {X 179.5126, Y 53.7103, Z -3.8333, A 0.000, B 0.000, C 0.000 }
gfCNCPoint3[1569] = {X 180.4426, Y 54.0357, Z -3.8333, A 0.000, B 0.000, C 0.000 }
gfCNCPoint3[1570] = {X 181.2769, Y 54.5599, Z -3.8333, A 0.000, B 0.000, C 0.000 }
gfCNCPoint3[1571] = {X 181.9736, Y 55.2566, Z -3.8333, A 0.000, B 0.000, C 0.000 }
gfCNCPoint3[1572] = {X 182.4978, Y 56.0909, Z -3.8333, A 0.000, B 0.000, C 0.000 }
gfCNCPoint3[1573] = {X 182.8232, Y 57.0209, Z -3.8333, A 0.000, B 0.000, C 0.000 }
gfCNCPoint3[1574] = {X 182.9335, Y 58.0000, Z -3.8333, A 0.000, B 0.000, C 0.000 }
gfCNCPoint3[1575] = {X 182.9334, Y 58.9704, Z -3.8333, A 0.000, B 0.000, C 0.000 }
gfCNCPoint3[1576] = {X 182.8587, Y 59.7419, Z -3.8333, A 0.000, B 0.000, C 0.000 }
gfCNCPoint3[1577] = {X 182.6499, Y 60.4883, Z -3.8333, A 0.000, B 0.000, C 0.000 }
gfCNCPoint3[1578] = {X 182.3133, Y 61.1865, Z -3.8333, A 0.000, B 0.000, C 0.000 }
gfCNCPoint3[1579] = {X 209.5374, Y 90.9000, Z -3.8333, A 0.000, B 0.000, C 0.000 }
gfCNCPoint3[1580] = {X 210.1907, Y 91.5629, Z -3.8333, A 0.000, B 0.000, C 0.000 }
gfCNCPoint3[1581] = {X 210.8906, Y 92.1765, Z -3.8333, A 0.000, B 0.000, C 0.000 }
gfCNCPoint3[1582] = {X 211.1522, Y 92.3414, Z -3.8333, A 0.000, B 0.000, C 0.000 }
gfCNCPoint3[1583] = {X 211.4457, Y 92.4390, Z -3.8333, A 0.000, B 0.000, C 0.000 }
gfCNCPoint3[1584] = {X 212.1215, Y 92.5835, Z -3.8333, A 0.000, B 0.000, C 0.000 }
gfCNCPoint3[1585] = {X 213.4015, Y 92.7447, Z -3.8333, A 0.000, B 0.000, C 0.000 }
gfCNCPoint3[1586] = {X 214.4547, Y 92.6560, Z -3.8333, A 0.000, B 0.000, C 0.000 }
gfCNCPoint3[1587] = {X 215.5099, Y 92.5958, Z -3.8333, A 0.000, B 0.000, C 0.000 }
gfCNCPoint3[1588] = {X 216.1640, Y 92.5237, Z -3.8333, A 0.000, B 0.000, C 0.000 }
gfCNCPoint3[1589] = {X 216.7937, Y 92.3330, Z -3.8333, A 0.000, B 0.000, C 0.000 }
gfCNCPoint3[1590] = {X 217.3778, Y 92.0300, Z -3.8333, A 0.000, B 0.000, C 0.000 }
gfCNCPoint3[1591] = {X 222.9188, Y 88.4542, Z -3.8333, A 0.000, B 0.000, C 0.000 }
gfCNCPoint3[1592] = {X 245.6531, Y 73.9167, Z -3.8333, A 0.000, B 0.000, C 0.000 }
gfCNCPoint3[1593] = {X 221.6008, Y 64.4777, Z -3.8333, A 0.000, B 0.000, C 0.000 }
gfCNCPoint3[1594] = {X 219.8423, Y 63.8889, Z -3.8333, A 0.000, B 0.000, C 0.000 }
gfCNCPoint3[1595] = {X 218.0279, Y 63.5052, Z -3.8333, A 0.000, B 0.000, C 0.000 }
gfCNCPoint3[1596] = {X 216.1816, Y 63.3315, Z -3.8333, A 0.000, B 0.000, C 0.000 }
gfCNCPoint3[1597] = {X 215.2274, Y 63.1935, Z -3.8333, A 0.000, B 0.000, C 0.000 }
gfCNCPoint3[1598] = {X 214.3262, Y 62.8509, Z -3.8333, A 0.000, B 0.000, C 0.000 }
gfCNCPoint3[1599] = {X 213.5213, Y 62.3203, Z -3.8333, A 0.000, B 0.000, C 0.000 }
gfCNCPoint3[1600] = {X 212.8512, Y 61.6271, Z -3.8333, A 0.000, B 0.000, C 0.000 }
gfCNCPoint3[1601] = {X 212.3482, Y 60.8046, Z -3.8333, A 0.000, B 0.000, C 0.000 }
gfCNCPoint3[1602] = {X 212.0364, Y 59.8923, Z -3.8333, A 0.000, B 0.000, C 0.000 }
gfCNCPoint3[1603] = {X 211.9308, Y 58.9340, Z -3.8333, A 0.000, B 0.000, C 0.000 }
gfCNCPoint3[1604] = {X 211.9308, Y 58.0000, Z -3.8333, A 0.000, B 0.000, C 0.000 }
gfCNCPoint3[1605] = {X 212.0411, Y 57.0209, Z -3.8333, A 0.000, B 0.000, C 0.000 }
gfCNCPoint3[1606] = {X 212.3665, Y 56.0909, Z -3.8333, A 0.000, B 0.000, C 0.000 }
gfCNCPoint3[1607] = {X 212.8907, Y 55.2566, Z -3.8333, A 0.000, B 0.000, C 0.000 }
gfCNCPoint3[1608] = {X 213.5875, Y 54.5599, Z -3.8333, A 0.000, B 0.000, C 0.000 }
gfCNCPoint3[1609] = {X 214.4217, Y 54.0357, Z -3.8333, A 0.000, B 0.000, C 0.000 }
gfCNCPoint3[1610] = {X 215.3517, Y 53.7103, Z -3.8333, A 0.000, B 0.000, C 0.000 }
gfCNCPoint3[1611] = {X 216.3308, Y 53.6000, Z -3.8333, A 0.000, B 0.000, C 0.000 }
gfCNCPoint3[1612] = {X 237.2617, Y 53.6000, Z -3.8333, A 0.000, B 0.000, C 0.000 }
gfCNCPoint3[1613] = {X 238.2408, Y 53.7103, Z -3.8333, A 0.000, B 0.000, C 0.000 }
gfCNCPoint3[1614] = {X 239.1708, Y 54.0357, Z -3.8333, A 0.000, B 0.000, C 0.000 }
gfCNCPoint3[1615] = {X 240.0050, Y 54.5599, Z -3.8333, A 0.000, B 0.000, C 0.000 }
gfCNCPoint3[1616] = {X 240.7017, Y 55.2566, Z -3.8333, A 0.000, B 0.000, C 0.000 }
gfCNCPoint3[1617] = {X 241.2260, Y 56.0909, Z -3.8333, A 0.000, B 0.000, C 0.000 }
gfCNCPoint3[1618] = {X 241.5514, Y 57.0209, Z -3.8333, A 0.000, B 0.000, C 0.000 }
gfCNCPoint3[1619] = {X 241.6617, Y 58.0000, Z -3.8333, A 0.000, B 0.000, C 0.000 }
gfCNCPoint3[1620] = {X 241.6617, Y 58.1778, Z -3.8333, A 0.000, B 0.000, C 0.000 }
gfCNCPoint3[1621] = {X 247.5187, Y 60.4610, Z -3.8333, A 0.000, B 0.000, C 0.000 }
gfCNCPoint3[1622] = {X 275.5531, Y 71.5846, Z -3.8333, A 0.000, B 0.000, C 0.000 }
gfCNCPoint3[1623] = {X 275.5525, Y 63.2812, Z -3.8333, A 0.000, B 0.000, C 0.000 }
gfCNCPoint3[1624] = {X 274.6933, Y 63.0560, Z -3.8333, A 0.000, B 0.000, C 0.000 }
gfCNCPoint3[1625] = {X 273.8967, Y 62.6628, Z -3.8333, A 0.000, B 0.000, C 0.000 }
gfCNCPoint3[1626] = {X 273.1954, Y 62.1176, Z -3.8333, A 0.000, B 0.000, C 0.000 }
gfCNCPoint3[1627] = {X 272.6179, Y 61.4427, Z -3.8333, A 0.000, B 0.000, C 0.000 }
gfCNCPoint3[1628] = {X 272.1877, Y 60.6655, Z -3.8333, A 0.000, B 0.000, C 0.000 }
gfCNCPoint3[1629] = {X 271.9224, Y 59.8178, Z -3.8333, A 0.000, B 0.000, C 0.000 }
gfCNCPoint3[1630] = {X 271.8327, Y 58.9340, Z -3.8333, A 0.000, B 0.000, C 0.000 }
gfCNCPoint3[1631] = {X 271.8327, Y 58.0000, Z -3.8333, A 0.000, B 0.000, C 0.000 }
gfCNCPoint3[1632] = {X 271.9430, Y 57.0209, Z -3.8333, A 0.000, B 0.000, C 0.000 }
gfCNCPoint3[1633] = {X 272.2684, Y 56.0909, Z -3.8333, A 0.000, B 0.000, C 0.000 }
gfCNCPoint3[1634] = {X 272.7926, Y 55.2566, Z -3.8333, A 0.000, B 0.000, C 0.000 }
gfCNCPoint3[1635] = {X 273.4893, Y 54.5599, Z -3.8333, A 0.000, B 0.000, C 0.000 }
gfCNCPoint3[1636] = {X 274.3236, Y 54.0357, Z -3.8333, A 0.000, B 0.000, C 0.000 }
gfCNCPoint3[1637] = {X 275.2536, Y 53.7103, Z -3.8333, A 0.000, B 0.000, C 0.000 }
gfCNCPoint3[1638] = {X 276.2327, Y 53.6000, Z -3.8333, A 0.000, B 0.000, C 0.000 }
gfCNCPoint3[1639] = {X 292.7731, Y 53.6000, Z -3.8333, A 0.000, B 0.000, C 0.000 }
gfCNCPoint3[1640] = {X 293.7522, Y 53.7103, Z -3.8333, A 0.000, B 0.000, C 0.000 }
gfCNCPoint3[1641] = {X 294.6822, Y 54.0357, Z -3.8333, A 0.000, B 0.000, C 0.000 }
gfCNCPoint3[1642] = {X 295.5164, Y 54.5599, Z -3.8333, A 0.000, B 0.000, C 0.000 }
gfCNCPoint3[1643] = {X 296.2131, Y 55.2566, Z -3.8333, A 0.000, B 0.000, C 0.000 }
gfCNCPoint3[1644] = {X 296.7373, Y 56.0909, Z -3.8333, A 0.000, B 0.000, C 0.000 }
gfCNCPoint3[1645] = {X 297.0628, Y 57.0209, Z -3.8333, A 0.000, B 0.000, C 0.000 }
gfCNCPoint3[1646] = {X 297.1731, Y 58.0000, Z -3.8333, A 0.000, B 0.000, C 0.000 }
gfCNCPoint3[1647] = {X 297.1731, Y 58.9354, Z -3.8333, A 0.000, B 0.000, C 0.000 }
gfCNCPoint3[1648] = {X 297.0810, Y 59.8183, Z -3.8333, A 0.000, B 0.000, C 0.000 }
gfCNCPoint3[1649] = {X 296.8143, Y 60.6650, Z -3.8333, A 0.000, B 0.000, C 0.000 }
gfCNCPoint3[1650] = {X 296.3836, Y 61.4412, Z -3.8333, A 0.000, B 0.000, C 0.000 }
gfCNCPoint3[1651] = {X 295.8063, Y 62.1157, Z -3.8333, A 0.000, B 0.000, C 0.000 }
gfCNCPoint3[1652] = {X 295.1059, Y 62.6610, Z -3.8333, A 0.000, B 0.000, C 0.000 }
gfCNCPoint3[1653] = {X 294.3106, Y 63.0553, Z -3.8333, A 0.000, B 0.000, C 0.000 }
gfCNCPoint3[1654] = {X 293.4524, Y 63.2826, Z -3.8333, A 0.000, B 0.000, C 0.000 }
gfCNCPoint3[1655] = {X 293.4524, Y 92.7111, Z -3.8333, A 0.000, B 0.000, C 0.000 }
gfCNCPoint3[1656] = {X 294.3104, Y 92.9409, Z -3.8333, A 0.000, B 0.000, C 0.000 }
gfCNCPoint3[1657] = {X 295.1052, Y 93.3371, Z -3.8333, A 0.000, B 0.000, C 0.000 }
gfCNCPoint3[1658] = {X 295.8052, Y 93.8838, Z -3.8333, A 0.000, B 0.000, C 0.000 }
gfCNCPoint3[1659] = {X 296.3821, Y 94.5591, Z -3.8333, A 0.000, B 0.000, C 0.000 }
gfCNCPoint3[1660] = {X 296.8128, Y 95.3358, Z -3.8333, A 0.000, B 0.000, C 0.000 }
gfCNCPoint3[1661] = {X 297.0801, Y 96.1828, Z -3.8333, A 0.000, B 0.000, C 0.000 }
gfCNCPoint3[1662] = {X 297.1731, Y 97.0661, Z -3.8333, A 0.000, B 0.000, C 0.000 }
gfCNCPoint3[1663] = {X 297.1731, Y 97.6950, Z -3.8333, A 0.000, B 0.000, C 0.000 }
gfCNCPoint3[1664] = {X 297.6531, Y 97.6950, Z -3.8333, A 0.000, B 0.000, C 0.000 }
gfCNCPoint3[1665] = {X 314.2152, Y 97.6950, Z -3.8333, A 0.000, B 0.000, C 0.000 }
gfCNCPoint3[1666] = {X 313.0165, Y 96.8444, Z -3.8333, A 0.000, B 0.000, C 0.000 }
gfCNCPoint3[1667] = {X 311.8817, Y 95.9102, Z -3.8333, A 0.000, B 0.000, C 0.000 }
gfCNCPoint3[1668] = {X 310.9060, Y 94.9484, Z -3.8333, A 0.000, B 0.000, C 0.000 }
gfCNCPoint3[1669] = {X 310.0417, Y 93.8854, Z -3.8333, A 0.000, B 0.000, C 0.000 }
gfCNCPoint3[1670] = {X 309.2077, Y 92.5708, Z -3.8333, A 0.000, B 0.000, C 0.000 }
gfCNCPoint3[1671] = {X 308.5440, Y 91.1625, Z -3.8333, A 0.000, B 0.000, C 0.000 }
gfCNCPoint3[1672] = {X 308.0608, Y 89.6825, Z -3.8333, A 0.000, B 0.000, C 0.000 }
gfCNCPoint3[1673] = {X 307.7074, Y 88.0127, Z -3.8333, A 0.000, B 0.000, C 0.000 }
gfCNCPoint3[1674] = {X 307.4985, Y 86.3187, Z -3.8333, A 0.000, B 0.000, C 0.000 }
gfCNCPoint3[1675] = {X 307.4357, Y 84.6130, Z -3.8333, A 0.000, B 0.000, C 0.000 }
gfCNCPoint3[1676] = {X 307.4369, Y 63.6744, Z -3.8333, A 0.000, B 0.000, C 0.000 }
gfCNCPoint3[1677] = {X 306.4284, Y 63.3062, Z -3.8333, A 0.000, B 0.000, C 0.000 }
gfCNCPoint3[1678] = {X 305.5249, Y 62.7263, Z -3.8333, A 0.000, B 0.000, C 0.000 }
gfCNCPoint3[1679] = {X 304.7700, Y 61.9630, Z -3.8333, A 0.000, B 0.000, C 0.000 }
gfCNCPoint3[1680] = {X 304.2002, Y 61.0530, Z -3.8333, A 0.000, B 0.000, C 0.000 }
gfCNCPoint3[1681] = {X 303.8433, Y 60.0404, Z -3.8333, A 0.000, B 0.000, C 0.000 }
gfCNCPoint3[1682] = {X 303.7164, Y 58.9744, Z -3.8333, A 0.000, B 0.000, C 0.000 }
gfCNCPoint3[1683] = {X 303.7162, Y 58.0000, Z -3.8333, A 0.000, B 0.000, C 0.000 }
gfCNCPoint3[1684] = {X 303.8100, Y 57.0480, Z -3.8333, A 0.000, B 0.000, C 0.000 }
gfCNCPoint3[1685] = {X 304.0877, Y 56.1325, Z -3.8333, A 0.000, B 0.000, C 0.000 }
gfCNCPoint3[1686] = {X 304.5387, Y 55.2888, Z -3.8333, A 0.000, B 0.000, C 0.000 }
gfCNCPoint3[1687] = {X 305.1455, Y 54.5493, Z -3.8333, A 0.000, B 0.000, C 0.000 }
gfCNCPoint3[1688] = {X 305.8850, Y 53.9424, Z -3.8333, A 0.000, B 0.000, C 0.000 }
gfCNCPoint3[1689] = {X 306.7287, Y 53.4915, Z -3.8333, A 0.000, B 0.000, C 0.000 }
gfCNCPoint3[1690] = {X 307.6442, Y 53.2138, Z -3.8333, A 0.000, B 0.000, C 0.000 }
gfCNCPoint3[1691] = {X 308.5962, Y 53.1200, Z -3.8333, A 0.000, B 0.000, C 0.000 }
gfCNCPoint3[1692] = {X 324.3107, Y 53.1200, Z -3.8333, A 0.000, B 0.000, C 0.000 }
gfCNCPoint3[1693] = {X 325.2627, Y 53.2138, Z -3.8333, A 0.000, B 0.000, C 0.000 }
gfCNCPoint3[1694] = {X 326.1782, Y 53.4915, Z -3.8333, A 0.000, B 0.000, C 0.000 }
gfCNCPoint3[1695] = {X 327.0219, Y 53.9424, Z -3.8333, A 0.000, B 0.000, C 0.000 }
gfCNCPoint3[1696] = {X 327.7614, Y 54.5493, Z -3.8333, A 0.000, B 0.000, C 0.000 }
gfCNCPoint3[1697] = {X 328.3683, Y 55.2888, Z -3.8333, A 0.000, B 0.000, C 0.000 }
gfCNCPoint3[1698] = {X 328.8192, Y 56.1325, Z -3.8333, A 0.000, B 0.000, C 0.000 }
gfCNCPoint3[1699] = {X 329.0969, Y 57.0480, Z -3.8333, A 0.000, B 0.000, C 0.000 }
gfCNCPoint3[1700] = {X 329.1907, Y 58.0000, Z -3.8333, A 0.000, B 0.000, C 0.000 }
gfCNCPoint3[1701] = {X 329.1907, Y 58.9341, Z -3.8333, A 0.000, B 0.000, C 0.000 }
gfCNCPoint3[1702] = {X 329.0670, Y 60.0067, Z -3.8333, A 0.000, B 0.000, C 0.000 }
gfCNCPoint3[1703] = {X 328.7123, Y 61.0264, Z -3.8333, A 0.000, B 0.000, C 0.000 }
gfCNCPoint3[1704] = {X 328.1437, Y 61.9442, Z -3.8333, A 0.000, B 0.000, C 0.000 }
gfCNCPoint3[1705] = {X 327.3885, Y 62.7159, Z -3.8333, A 0.000, B 0.000, C 0.000 }
gfCNCPoint3[1706] = {X 326.4832, Y 63.3042, Z -3.8333, A 0.000, B 0.000, C 0.000 }
gfCNCPoint3[1707] = {X 325.4713, Y 63.6808, Z -3.8333, A 0.000, B 0.000, C 0.000 }
gfCNCPoint3[1708] = {X 325.4729, Y 83.2269, Z -3.8333, A 0.000, B 0.000, C 0.000 }
gfCNCPoint3[1709] = {X 325.4864, Y 84.6073, Z -3.8333, A 0.000, B 0.000, C 0.000 }
gfCNCPoint3[1710] = {X 325.5523, Y 85.7201, Z -3.8333, A 0.000, B 0.000, C 0.000 }
gfCNCPoint3[1711] = {X 325.7425, Y 86.8185, Z -3.8333, A 0.000, B 0.000, C 0.000 }
gfCNCPoint3[1712] = {X 325.8865, Y 86.9527, Z -3.8333, A 0.000, B 0.000, C 0.000 }
gfCNCPoint3[1713] = {X 326.0548, Y 87.0548, Z -3.8333, A 0.000, B 0.000, C 0.000 }
gfCNCPoint3[1714] = {X 326.4834, Y 87.2970, Z -3.8333, A 0.000, B 0.000, C 0.000 }
gfCNCPoint3[1715] = {X 327.8568, Y 87.8654, Z -3.8333, A 0.000, B 0.000, C 0.000 }
gfCNCPoint3[1716] = {X 329.2840, Y 88.2810, Z -3.8333, A 0.000, B 0.000, C 0.000 }
gfCNCPoint3[1717] = {X 332.3217, Y 88.8893, Z -3.8333, A 0.000, B 0.000, C 0.000 }
gfCNCPoint3[1718] = {X 335.3954, Y 89.2773, Z -3.8333, A 0.000, B 0.000, C 0.000 }
gfCNCPoint3[1719] = {X 339.5149, Y 89.5962, Z -3.8333, A 0.000, B 0.000, C 0.000 }
gfCNCPoint3[1720] = {X 343.6430, Y 89.7751, Z -3.8333, A 0.000, B 0.000, C 0.000 }
gfCNCPoint3[1721] = {X 347.7747, Y 89.8137, Z -3.8333, A 0.000, B 0.000, C 0.000 }
gfCNCPoint3[1722] = {X 352.1398, Y 89.7758, Z -3.8333, A 0.000, B 0.000, C 0.000 }
gfCNCPoint3[1723] = {X 356.5008, Y 89.5808, Z -3.8333, A 0.000, B 0.000, C 0.000 }
gfCNCPoint3[1724] = {X 360.8519, Y 89.2291, Z -3.8333, A 0.000, B 0.000, C 0.000 }
gfCNCPoint3[1725] = {X 363.1336, Y 88.9455, Z -3.8333, A 0.000, B 0.000, C 0.000 }
gfCNCPoint3[1726] = {X 365.3941, Y 88.5252, Z -3.8333, A 0.000, B 0.000, C 0.000 }
gfCNCPoint3[1727] = {X 367.6253, Y 87.9697, Z -3.8333, A 0.000, B 0.000, C 0.000 }
gfCNCPoint3[1728] = {X 368.9187, Y 87.4948, Z -3.8333, A 0.000, B 0.000, C 0.000 }
gfCNCPoint3[1729] = {X 370.1143, Y 86.8098, Z -3.8333, A 0.000, B 0.000, C 0.000 }
gfCNCPoint3[1730] = {X 370.2988, Y 85.3241, Z -3.8333, A 0.000, B 0.000, C 0.000 }
gfCNCPoint3[1731] = {X 370.3604, Y 83.8282, Z -3.8333, A 0.000, B 0.000, C 0.000 }
gfCNCPoint3[1732] = {X 370.3589, Y 63.6741, Z -3.8333, A 0.000, B 0.000, C 0.000 }
gfCNCPoint3[1733] = {X 369.3507, Y 63.3057, Z -3.8333, A 0.000, B 0.000, C 0.000 }
gfCNCPoint3[1734] = {X 368.4474, Y 62.7259, Z -3.8333, A 0.000, B 0.000, C 0.000 }
gfCNCPoint3[1735] = {X 367.6927, Y 61.9625, Z -3.8333, A 0.000, B 0.000, C 0.000 }
gfCNCPoint3[1736] = {X 367.1231, Y 61.0526, Z -3.8333, A 0.000, B 0.000, C 0.000 }
gfCNCPoint3[1737] = {X 366.7663, Y 60.0403, Z -3.8333, A 0.000, B 0.000, C 0.000 }
gfCNCPoint3[1738] = {X 366.6394, Y 58.9744, Z -3.8333, A 0.000, B 0.000, C 0.000 }
gfCNCPoint3[1739] = {X 366.6393, Y 58.0000, Z -3.8333, A 0.000, B 0.000, C 0.000 }
gfCNCPoint3[1740] = {X 366.7331, Y 57.0480, Z -3.8333, A 0.000, B 0.000, C 0.000 }
gfCNCPoint3[1741] = {X 367.0108, Y 56.1325, Z -3.8333, A 0.000, B 0.000, C 0.000 }
gfCNCPoint3[1742] = {X 367.4617, Y 55.2888, Z -3.8333, A 0.000, B 0.000, C 0.000 }
gfCNCPoint3[1743] = {X 368.0686, Y 54.5493, Z -3.8333, A 0.000, B 0.000, C 0.000 }
gfCNCPoint3[1744] = {X 368.8081, Y 53.9424, Z -3.8333, A 0.000, B 0.000, C 0.000 }
gfCNCPoint3[1745] = {X 369.6518, Y 53.4915, Z -3.8333, A 0.000, B 0.000, C 0.000 }
gfCNCPoint3[1746] = {X 370.5672, Y 53.2138, Z -3.8333, A 0.000, B 0.000, C 0.000 }
gfCNCPoint3[1747] = {X 371.5193, Y 53.1200, Z -3.8333, A 0.000, B 0.000, C 0.000 }
gfCNCPoint3[1748] = {X 388.0597, Y 53.1200, Z -3.8333, A 0.000, B 0.000, C 0.000 }
gfCNCPoint3[1749] = {X 389.0355, Y 53.2186, Z -3.8333, A 0.000, B 0.000, C 0.000 }
gfCNCPoint3[1750] = {X 389.9719, Y 53.5102, Z -3.8333, A 0.000, B 0.000, C 0.000 }
gfCNCPoint3[1751] = {X 390.8310, Y 53.9833, Z -3.8333, A 0.000, B 0.000, C 0.000 }
gfCNCPoint3[1752] = {X 391.5783, Y 54.6186, Z -3.8333, A 0.000, B 0.000, C 0.000 }
gfCNCPoint3[1753] = {X 392.1572, Y 55.3496, Z -3.8333, A 0.000, B 0.000, C 0.000 }
gfCNCPoint3[1754] = {X 392.5865, Y 56.1774, Z -3.8333, A 0.000, B 0.000, C 0.000 }
gfCNCPoint3[1755] = {X 392.8506, Y 57.0718, Z -3.8333, A 0.000, B 0.000, C 0.000 }
gfCNCPoint3[1756] = {X 392.9397, Y 58.0000, Z -3.8333, A 0.000, B 0.000, C 0.000 }
gfCNCPoint3[1757] = {X 392.9395, Y 58.9743, Z -3.8333, A 0.000, B 0.000, C 0.000 }
gfCNCPoint3[1758] = {X 392.8779, Y 59.7081, Z -3.8333, A 0.000, B 0.000, C 0.000 }
gfCNCPoint3[1759] = {X 392.7066, Y 60.4243, Z -3.8333, A 0.000, B 0.000, C 0.000 }
gfCNCPoint3[1760] = {X 392.4294, Y 61.1066, Z -3.8333, A 0.000, B 0.000, C 0.000 }
gfCNCPoint3[1761] = {X 392.0494, Y 61.7445, Z -3.8333, A 0.000, B 0.000, C 0.000 }
gfCNCPoint3[1762] = {X 391.5775, Y 62.3177, Z -3.8333, A 0.000, B 0.000, C 0.000 }
gfCNCPoint3[1763] = {X 390.8818, Y 62.9185, Z -3.8333, A 0.000, B 0.000, C 0.000 }
gfCNCPoint3[1764] = {X 390.0862, Y 63.3787, Z -3.8333, A 0.000, B 0.000, C 0.000 }
gfCNCPoint3[1765] = {X 389.2186, Y 63.6824, Z -3.8333, A 0.000, B 0.000, C 0.000 }
gfCNCPoint3[1766] = {X 389.2177, Y 73.4812, Z -3.8333, A 0.000, B 0.000, C 0.000 }
gfCNCPoint3[1767] = {X 398.8177, Y 73.4821, Z -3.8333, A 0.000, B 0.000, C 0.000 }
gfCNCPoint3[1768] = {X 398.8170, Y 80.5583, Z -3.8333, A 0.000, B 0.000, C 0.000 }
gfCNCPoint3[1769] = {X 405.8042, Y 76.0834, Z -3.8333, A 0.000, B 0.000, C 0.000 }
gfCNCPoint3[1770] = {X 400.0367, Y 73.8205, Z -3.8333, A 0.000, B 0.000, C 0.000 }
gfCNCPoint3[1771] = {X 399.4360, Y 73.6196, Z -3.8333, A 0.000, B 0.000, C 0.000 }
gfCNCPoint3[1772] = {X 398.8177, Y 73.4821, Z -3.8333, A 0.000, B 0.000, C 0.000 }
gfCNCPoint3[1773] = {X 396.4177, Y 73.4819, Z -3.8333, A 0.000, B 0.000, C 0.000 }
gfCNCPoint3[1774] = {X 396.4166, Y 84.5897, Z -3.8333, A 0.000, B 0.000, C 0.000 }
gfCNCPoint3[1775] = {X 396.4165, Y 84.9457, Z -3.8333, A 0.000, B 0.000, C 0.000 }
gfCNCPoint3[1776] = {X 411.0600, Y 75.5674, Z -3.8333, A 0.000, B 0.000, C 0.000 }
gfCNCPoint3[1777] = {X 400.9153, Y 71.5871, Z -3.8333, A 0.000, B 0.000, C 0.000 }
gfCNCPoint3[1778] = {X 399.6205, Y 71.1936, Z -3.8333, A 0.000, B 0.000, C 0.000 }
gfCNCPoint3[1779] = {X 398.2797, Y 71.0109, Z -3.8333, A 0.000, B 0.000, C 0.000 }
gfCNCPoint3[1780] = {X 397.3452, Y 70.9531, Z -3.8333, A 0.000, B 0.000, C 0.000 }
gfCNCPoint3[1781] = {X 396.4179, Y 70.8230, Z -3.8333, A 0.000, B 0.000, C 0.000 }
gfCNCPoint3[1782] = {X 396.4177, Y 73.4819, Z -3.8333, A 0.000, B 0.000, C 0.000 }
gfCNCPoint3[1783] = {X 394.0177, Y 73.4817, Z -3.8333, A 0.000, B 0.000, C 0.000 }
gfCNCPoint3[1784] = {X 394.0166, Y 84.5974, Z -3.8333, A 0.000, B 0.000, C 0.000 }
gfCNCPoint3[1785] = {X 394.0171, Y 84.7631, Z -3.8333, A 0.000, B 0.000, C 0.000 }
gfCNCPoint3[1786] = {X 394.0166, Y 84.9289, Z -3.8333, A 0.000, B 0.000, C 0.000 }
gfCNCPoint3[1787] = {X 393.9662, Y 86.3339, Z -3.8333, A 0.000, B 0.000, C 0.000 }
gfCNCPoint3[1788] = {X 393.8348, Y 87.7336, Z -3.8333, A 0.000, B 0.000, C 0.000 }
gfCNCPoint3[1789] = {X 395.0962, Y 87.4749, Z -3.8333, A 0.000, B 0.000, C 0.000 }
gfCNCPoint3[1790] = {X 396.3809, Y 87.3860, Z -3.8333, A 0.000, B 0.000, C 0.000 }
gfCNCPoint3[1791] = {X 396.7496, Y 87.3712, Z -3.8333, A 0.000, B 0.000, C 0.000 }
gfCNCPoint3[1792] = {X 397.1178, Y 87.3466, Z -3.8333, A 0.000, B 0.000, C 0.000 }
gfCNCPoint3[1793] = {X 416.3157, Y 75.0514, Z -3.8333, A 0.000, B 0.000, C 0.000 }
gfCNCPoint3[1794] = {X 401.7938, Y 69.3536, Z -3.8333, A 0.000, B 0.000, C 0.000 }
gfCNCPoint3[1795] = {X 400.6813, Y 68.9838, Z -3.8333, A 0.000, B 0.000, C 0.000 }
gfCNCPoint3[1796] = {X 399.5354, Y 68.7357, Z -3.8333, A 0.000, B 0.000, C 0.000 }
gfCNCPoint3[1797] = {X 398.3696, Y 68.6122, Z -3.8333, A 0.000, B 0.000, C 0.000 }
gfCNCPoint3[1798] = {X 397.6033, Y 68.5669, Z -3.8333, A 0.000, B 0.000, C 0.000 }
gfCNCPoint3[1799] = {X 396.8431, Y 68.4610, Z -3.8333, A 0.000, B 0.000, C 0.000 }
gfCNCPoint3[1800] = {X 395.3927, Y 68.0820, Z -3.8333, A 0.000, B 0.000, C 0.000 }
gfCNCPoint3[1801] = {X 394.0183, Y 67.4837, Z -3.8333, A 0.000, B 0.000, C 0.000 }
gfCNCPoint3[1802] = {X 394.0177, Y 73.4817, Z -3.8333, A 0.000, B 0.000, C 0.000 }
gfCNCPoint3[1803] = {X 391.6177, Y 73.4814, Z -3.8333, A 0.000, B 0.000, C 0.000 }
gfCNCPoint3[1804] = {X 391.6166, Y 84.6054, Z -3.8333, A 0.000, B 0.000, C 0.000 }
gfCNCPoint3[1805] = {X 391.5806, Y 86.0256, Z -3.8333, A 0.000, B 0.000, C 0.000 }
gfCNCPoint3[1806] = {X 391.4528, Y 87.4406, Z -3.8333, A 0.000, B 0.000, C 0.000 }
gfCNCPoint3[1807] = {X 391.2285, Y 88.8722, Z -3.8333, A 0.000, B 0.000, C 0.000 }
gfCNCPoint3[1808] = {X 390.9103, Y 90.2860, Z -3.8333, A 0.000, B 0.000, C 0.000 }
gfCNCPoint3[1809] = {X 390.3341, Y 92.0499, Z -3.8333, A 0.000, B 0.000, C 0.000 }
gfCNCPoint3[1810] = {X 389.5427, Y 93.7283, Z -3.8333, A 0.000, B 0.000, C 0.000 }
gfCNCPoint3[1811] = {X 388.5483, Y 95.2950, Z -3.8333, A 0.000, B 0.000, C 0.000 }
gfCNCPoint3[1812] = {X 389.3446, Y 95.2950, Z -3.8333, A 0.000, B 0.000, C 0.000 }
gfCNCPoint3[1813] = {X 389.7639, Y 94.0857, Z -3.8333, A 0.000, B 0.000, C 0.000 }
gfCNCPoint3[1814] = {X 390.3885, Y 92.9685, Z -3.8333, A 0.000, B 0.000, C 0.000 }
gfCNCPoint3[1815] = {X 391.1991, Y 91.9780, Z -3.8333, A 0.000, B 0.000, C 0.000 }
gfCNCPoint3[1816] = {X 392.1706, Y 91.1448, Z -3.8333, A 0.000, B 0.000, C 0.000 }
gfCNCPoint3[1817] = {X 393.2730, Y 90.4945, Z -3.8333, A 0.000, B 0.000, C 0.000 }
gfCNCPoint3[1818] = {X 394.4723, Y 90.0474, Z -3.8333, A 0.000, B 0.000, C 0.000 }
gfCNCPoint3[1819] = {X 395.4337, Y 89.8512, Z -3.8333, A 0.000, B 0.000, C 0.000 }
gfCNCPoint3[1820] = {X 396.4127, Y 89.7859, Z -3.8333, A 0.000, B 0.000, C 0.000 }
gfCNCPoint3[1821] = {X 397.1772, Y 89.7464, Z -3.8333, A 0.000, B 0.000, C 0.000 }
gfCNCPoint3[1822] = {X 397.9389, Y 89.6707, Z -3.8333, A 0.000, B 0.000, C 0.000 }
gfCNCPoint3[1823] = {X 421.5715, Y 74.5354, Z -3.8333, A 0.000, B 0.000, C 0.000 }
gfCNCPoint3[1824] = {X 402.6723, Y 67.1202, Z -3.8333, A 0.000, B 0.000, C 0.000 }
gfCNCPoint3[1825] = {X 401.3007, Y 66.6651, Z -3.8333, A 0.000, B 0.000, C 0.000 }
gfCNCPoint3[1826] = {X 399.8878, Y 66.3616, Z -3.8333, A 0.000, B 0.000, C 0.000 }
gfCNCPoint3[1827] = {X 398.4502, Y 66.2133, Z -3.8333, A 0.000, B 0.000, C 0.000 }
gfCNCPoint3[1828] = {X 397.3057, Y 66.1056, Z -3.8333, A 0.000, B 0.000, C 0.000 }
gfCNCPoint3[1829] = {X 396.1924, Y 65.8191, Z -3.8333, A 0.000, B 0.000, C 0.000 }
gfCNCPoint3[1830] = {X 395.1381, Y 65.3609, Z -3.8333, A 0.000, B 0.000, C 0.000 }
gfCNCPoint3[1831] = {X 394.1690, Y 64.7425, Z -3.8333, A 0.000, B 0.000, C 0.000 }
gfCNCPoint3[1832] = {X 393.3094, Y 63.9792, Z -3.8333, A 0.000, B 0.000, C 0.000 }
gfCNCPoint3[1833] = {X 392.5122, Y 64.6965, Z -3.8333, A 0.000, B 0.000, C 0.000 }
gfCNCPoint3[1834] = {X 391.6185, Y 65.2893, Z -3.8333, A 0.000, B 0.000, C 0.000 }
gfCNCPoint3[1835] = {X 391.6177, Y 73.4814, Z -3.8333, A 0.000, B 0.000, C 0.000 }
gfCNCPoint3[1836] = {X 389.2177, Y 73.4812, Z -3.8333, A 0.000, B 0.000, C 0.000 }
gfCNCPoint3[1837] = {X 389.2166, Y 84.6139, Z -3.8333, A 0.000, B 0.000, C 0.000 }
gfCNCPoint3[1838] = {X 389.1547, Y 86.3199, Z -3.8333, A 0.000, B 0.000, C 0.000 }
gfCNCPoint3[1839] = {X 388.9444, Y 88.0140, Z -3.8333, A 0.000, B 0.000, C 0.000 }
gfCNCPoint3[1840] = {X 388.5872, Y 89.6833, Z -3.8333, A 0.000, B 0.000, C 0.000 }
gfCNCPoint3[1841] = {X 388.1040, Y 91.1629, Z -3.8333, A 0.000, B 0.000, C 0.000 }
gfCNCPoint3[1842] = {X 387.4403, Y 92.5708, Z -3.8333, A 0.000, B 0.000, C 0.000 }
gfCNCPoint3[1843] = {X 386.6062, Y 93.8850, Z -3.8333, A 0.000, B 0.000, C 0.000 }
gfCNCPoint3[1844] = {X 385.8740, Y 94.7997, Z -3.8333, A 0.000, B 0.000, C 0.000 }
gfCNCPoint3[1845] = {X 385.0592, Y 95.6417, Z -3.8333, A 0.000, B 0.000, C 0.000 }
gfCNCPoint3[1846] = {X 383.7991, Y 96.7249, Z -3.8333, A 0.000, B 0.000, C 0.000 }
gfCNCPoint3[1847] = {X 382.4501, Y 97.6950, Z -3.8333, A 0.000, B 0.000, C 0.000 }
gfCNCPoint3[1848] = {X 382.1870, Y 97.2935, Z -3.8333, A 0.000, B 0.000, C 0.000 }
gfCNCPoint3[1849] = {X 381.0197, Y 97.9991, Z -3.8333, A 0.000, B 0.000, C 0.000 }
gfCNCPoint3[1850] = {X 379.8040, Y 98.6178, Z -3.8333, A 0.000, B 0.000, C 0.000 }
gfCNCPoint3[1851] = {X 377.5271, Y 99.5763, Z -3.8333, A 0.000, B 0.000, C 0.000 }
gfCNCPoint3[1852] = {X 375.1871, Y 100.3685, Z -3.8333, A 0.000, B 0.000, C 0.000 }
gfCNCPoint3[1853] = {X 372.7962, Y 100.9903, Z -3.8333, A 0.000, B 0.000, C 0.000 }
gfCNCPoint3[1854] = {X 368.9811, Y 101.7284, Z -3.8333, A 0.000, B 0.000, C 0.000 }
gfCNCPoint3[1855] = {X 365.1349, Y 102.2822, Z -3.8333, A 0.000, B 0.000, C 0.000 }
gfCNCPoint3[1856] = {X 361.2665, Y 102.6505, Z -3.8333, A 0.000, B 0.000, C 0.000 }
gfCNCPoint3[1857] = {X 355.1239, Y 102.9838, Z -3.8333, A 0.000, B 0.000, C 0.000 }
gfCNCPoint3[1858] = {X 348.9736, Y 103.1123, Z -3.8333, A 0.000, B 0.000, C 0.000 }
gfCNCPoint3[1859] = {X 342.8224, Y 103.0359, Z -3.8333, A 0.000, B 0.000, C 0.000 }
gfCNCPoint3[1860] = {X 336.6772, Y 102.7546, Z -3.8333, A 0.000, B 0.000, C 0.000 }
gfCNCPoint3[1861] = {X 333.1845, Y 102.4782, Z -3.8333, A 0.000, B 0.000, C 0.000 }
gfCNCPoint3[1862] = {X 329.7053, Y 102.0649, Z -3.8333, A 0.000, B 0.000, C 0.000 }
gfCNCPoint3[1863] = {X 326.2450, Y 101.5154, Z -3.8333, A 0.000, B 0.000, C 0.000 }
gfCNCPoint3[1864] = {X 323.3894, Y 100.9105, Z -3.8333, A 0.000, B 0.000, C 0.000 }
gfCNCPoint3[1865] = {X 320.5865, Y 100.0959, Z -3.8333, A 0.000, B 0.000, C 0.000 }
gfCNCPoint3[1866] = {X 317.8516, Y 99.0762, Z -3.8333, A 0.000, B 0.000, C 0.000 }
gfCNCPoint3[1867] = {X 316.3331, Y 98.3749, Z -3.8333, A 0.000, B 0.000, C 0.000 }
gfCNCPoint3[1868] = {X 314.8784, Y 97.5497, Z -3.8333, A 0.000, B 0.000, C 0.000 }
gfCNCPoint3[1869] = {X 313.4974, Y 96.6061, Z -3.8333, A 0.000, B 0.000, C 0.000 }
gfCNCPoint3[1870] = {X 312.1998, Y 95.5508, Z -3.8333, A 0.000, B 0.000, C 0.000 }
gfCNCPoint3[1871] = {X 311.1892, Y 94.5456, Z -3.8333, A 0.000, B 0.000, C 0.000 }
gfCNCPoint3[1872] = {X 310.3050, Y 93.4277, Z -3.8333, A 0.000, B 0.000, C 0.000 }
gfCNCPoint3[1873] = {X 309.5596, Y 92.2127, Z -3.8333, A 0.000, B 0.000, C 0.000 }
gfCNCPoint3[1874] = {X 308.9636, Y 90.9180, Z -3.8333, A 0.000, B 0.000, C 0.000 }
gfCNCPoint3[1875] = {X 308.5253, Y 89.5616, Z -3.8333, A 0.000, B 0.000, C 0.000 }
gfCNCPoint3[1876] = {X 308.1806, Y 87.9321, Z -3.8333, A 0.000, B 0.000, C 0.000 }
gfCNCPoint3[1877] = {X 307.9768, Y 86.2791, Z -3.8333, A 0.000, B 0.000, C 0.000 }
gfCNCPoint3[1878] = {X 307.9157, Y 84.6146, Z -3.8333, A 0.000, B 0.000, C 0.000 }
gfCNCPoint3[1879] = {X 307.9170, Y 63.2813, Z -3.8333, A 0.000, B 0.000, C 0.000 }
gfCNCPoint3[1880] = {X 307.0575, Y 63.0562, Z -3.8333, A 0.000, B 0.000, C 0.000 }
gfCNCPoint3[1881] = {X 306.2608, Y 62.6631, Z -3.8333, A 0.000, B 0.000, C 0.000 }
gfCNCPoint3[1882] = {X 305.5593, Y 62.1180, Z -3.8333, A 0.000, B 0.000, C 0.000 }
gfCNCPoint3[1883] = {X 304.9816, Y 61.4430, Z -3.8333, A 0.000, B 0.000, C 0.000 }
gfCNCPoint3[1884] = {X 304.5513, Y 60.6658, Z -3.8333, A 0.000, B 0.000, C 0.000 }
gfCNCPoint3[1885] = {X 304.2859, Y 59.8179, Z -3.8333, A 0.000, B 0.000, C 0.000 }
gfCNCPoint3[1886] = {X 304.1962, Y 58.9340, Z -3.8333, A 0.000, B 0.000, C 0.000 }
gfCNCPoint3[1887] = {X 304.1962, Y 58.0000, Z -3.8333, A 0.000, B 0.000, C 0.000 }
gfCNCPoint3[1888] = {X 304.3065, Y 57.0209, Z -3.8333, A 0.000, B 0.000, C 0.000 }
gfCNCPoint3[1889] = {X 304.6320, Y 56.0909, Z -3.8333, A 0.000, B 0.000, C 0.000 }
gfCNCPoint3[1890] = {X 305.1562, Y 55.2566, Z -3.8333, A 0.000, B 0.000, C 0.000 }
gfCNCPoint3[1891] = {X 305.8529, Y 54.5599, Z -3.8333, A 0.000, B 0.000, C 0.000 }
gfCNCPoint3[1892] = {X 306.6871, Y 54.0357, Z -3.8333, A 0.000, B 0.000, C 0.000 }
gfCNCPoint3[1893] = {X 307.6171, Y 53.7103, Z -3.8333, A 0.000, B 0.000, C 0.000 }
gfCNCPoint3[1894] = {X 308.5962, Y 53.6000, Z -3.8333, A 0.000, B 0.000, C 0.000 }
gfCNCPoint3[1895] = {X 324.3107, Y 53.6000, Z -3.8333, A 0.000, B 0.000, C 0.000 }
gfCNCPoint3[1896] = {X 325.2898, Y 53.7103, Z -3.8333, A 0.000, B 0.000, C 0.000 }
gfCNCPoint3[1897] = {X 326.2198, Y 54.0357, Z -3.8333, A 0.000, B 0.000, C 0.000 }
gfCNCPoint3[1898] = {X 327.0540, Y 54.5599, Z -3.8333, A 0.000, B 0.000, C 0.000 }
gfCNCPoint3[1899] = {X 327.7507, Y 55.2566, Z -3.8333, A 0.000, B 0.000, C 0.000 }
gfCNCPoint3[1900] = {X 328.2749, Y 56.0909, Z -3.8333, A 0.000, B 0.000, C 0.000 }
gfCNCPoint3[1901] = {X 328.6004, Y 57.0209, Z -3.8333, A 0.000, B 0.000, C 0.000 }
gfCNCPoint3[1902] = {X 328.7107, Y 58.0000, Z -3.8333, A 0.000, B 0.000, C 0.000 }
gfCNCPoint3[1903] = {X 328.7107, Y 58.9364, Z -3.8333, A 0.000, B 0.000, C 0.000 }
gfCNCPoint3[1904] = {X 328.6168, Y 59.8191, Z -3.8333, A 0.000, B 0.000, C 0.000 }
gfCNCPoint3[1905] = {X 328.3491, Y 60.6654, Z -3.8333, A 0.000, B 0.000, C 0.000 }
gfCNCPoint3[1906] = {X 327.9184, Y 61.4416, Z -3.8333, A 0.000, B 0.000, C 0.000 }
gfCNCPoint3[1907] = {X 327.3418, Y 62.1165, Z -3.8333, A 0.000, B 0.000, C 0.000 }
gfCNCPoint3[1908] = {X 326.6425, Y 62.6632, Z -3.8333, A 0.000, B 0.000, C 0.000 }
gfCNCPoint3[1909] = {X 325.8485, Y 63.0599, Z -3.8333, A 0.000, B 0.000, C 0.000 }
gfCNCPoint3[1910] = {X 324.9913, Y 63.2906, Z -3.8333, A 0.000, B 0.000, C 0.000 }
gfCNCPoint3[1911] = {X 324.9929, Y 83.2293, Z -3.8333, A 0.000, B 0.000, C 0.000 }
gfCNCPoint3[1912] = {X 325.0064, Y 84.6145, Z -3.8333, A 0.000, B 0.000, C 0.000 }
gfCNCPoint3[1913] = {X 325.0823, Y 85.8325, Z -3.8333, A 0.000, B 0.000, C 0.000 }
gfCNCPoint3[1914] = {X 325.3001, Y 87.0334, Z -3.8333, A 0.000, B 0.000, C 0.000 }
gfCNCPoint3[1915] = {X 325.5332, Y 87.2840, Z -3.8333, A 0.000, B 0.000, C 0.000 }
gfCNCPoint3[1916] = {X 325.8187, Y 87.4727, Z -3.8333, A 0.000, B 0.000, C 0.000 }
gfCNCPoint3[1917] = {X 326.2612, Y 87.7228, Z -3.8333, A 0.000, B 0.000, C 0.000 }
gfCNCPoint3[1918] = {X 327.6909, Y 88.3158, Z -3.8333, A 0.000, B 0.000, C 0.000 }
gfCNCPoint3[1919] = {X 329.1769, Y 88.7489, Z -3.8333, A 0.000, B 0.000, C 0.000 }
gfCNCPoint3[1920] = {X 332.2475, Y 89.3635, Z -3.8333, A 0.000, B 0.000, C 0.000 }
gfCNCPoint3[1921] = {X 335.3543, Y 89.7555, Z -3.8333, A 0.000, B 0.000, C 0.000 }
gfCNCPoint3[1922] = {X 339.4910, Y 90.0756, Z -3.8333, A 0.000, B 0.000, C 0.000 }
gfCNCPoint3[1923] = {X 343.6362, Y 90.2551, Z -3.8333, A 0.000, B 0.000, C 0.000 }
gfCNCPoint3[1924] = {X 347.7851, Y 90.2937, Z -3.8333, A 0.000, B 0.000, C 0.000 }
gfCNCPoint3[1925] = {X 352.1632, Y 90.2552, Z -3.8333, A 0.000, B 0.000, C 0.000 }
gfCNCPoint3[1926] = {X 356.5371, Y 90.0594, Z -3.8333, A 0.000, B 0.000, C 0.000 }
gfCNCPoint3[1927] = {X 360.9012, Y 89.7066, Z -3.8333, A 0.000, B 0.000, C 0.000 }
gfCNCPoint3[1928] = {X 363.2108, Y 89.4192, Z -3.8333, A 0.000, B 0.000, C 0.000 }
gfCNCPoint3[1929] = {X 365.4989, Y 88.9936, Z -3.8333, A 0.000, B 0.000, C 0.000 }
gfCNCPoint3[1930] = {X 367.7574, Y 88.4312, Z -3.8333, A 0.000, B 0.000, C 0.000 }
gfCNCPoint3[1931] = {X 368.6802, Y 88.1208, Z -3.8333, A 0.000, B 0.000, C 0.000 }
gfCNCPoint3[1932] = {X 369.5625, Y 87.7089, Z -3.8333, A 0.000, B 0.000, C 0.000 }
gfCNCPoint3[1933] = {X 370.3930, Y 87.2007, Z -3.8333, A 0.000, B 0.000, C 0.000 }
gfCNCPoint3[1934] = {X 370.5208, Y 87.0677, Z -3.8333, A 0.000, B 0.000, C 0.000 }
gfCNCPoint3[1935] = {X 370.5866, Y 86.8954, Z -3.8333, A 0.000, B 0.000, C 0.000 }
gfCNCPoint3[1936] = {X 370.7769, Y 85.3670, Z -3.8333, A 0.000, B 0.000, C 0.000 }
gfCNCPoint3[1937] = {X 370.8404, Y 83.8281, Z -3.8333, A 0.000, B 0.000, C 0.000 }
gfCNCPoint3[1938] = {X 370.8389, Y 63.2811, Z -3.8333, A 0.000, B 0.000, C 0.000 }
gfCNCPoint3[1939] = {X 369.9797, Y 63.0559, Z -3.8333, A 0.000, B 0.000, C 0.000 }
gfCNCPoint3[1940] = {X 369.1832, Y 62.6627, Z -3.8333, A 0.000, B 0.000, C 0.000 }
gfCNCPoint3[1941] = {X 368.4819, Y 62.1175, Z -3.8333, A 0.000, B 0.000, C 0.000 }
gfCNCPoint3[1942] = {X 367.9044, Y 61.4426, Z -3.8333, A 0.000, B 0.000, C 0.000 }
gfCNCPoint3[1943] = {X 367.4743, Y 60.6655, Z -3.8333, A 0.000, B 0.000, C 0.000 }
gfCNCPoint3[1944] = {X 367.2089, Y 59.8178, Z -3.8333, A 0.000, B 0.000, C 0.000 }
gfCNCPoint3[1945] = {X 367.1193, Y 58.9340, Z -3.8333, A 0.000, B 0.000, C 0.000 }
gfCNCPoint3[1946] = {X 367.1193, Y 58.0000, Z -3.8333, A 0.000, B 0.000, C 0.000 }
gfCNCPoint3[1947] = {X 367.2296, Y 57.0209, Z -3.8333, A 0.000, B 0.000, C 0.000 }
gfCNCPoint3[1948] = {X 367.5550, Y 56.0909, Z -3.8333, A 0.000, B 0.000, C 0.000 }
gfCNCPoint3[1949] = {X 368.0792, Y 55.2566, Z -3.8333, A 0.000, B 0.000, C 0.000 }
gfCNCPoint3[1950] = {X 368.7759, Y 54.5599, Z -3.8333, A 0.000, B 0.000, C 0.000 }
gfCNCPoint3[1951] = {X 369.6102, Y 54.0357, Z -3.8333, A 0.000, B 0.000, C 0.000 }
gfCNCPoint3[1952] = {X 370.5402, Y 53.7103, Z -3.8333, A 0.000, B 0.000, C 0.000 }
gfCNCPoint3[1953] = {X 371.5193, Y 53.6000, Z -3.8333, A 0.000, B 0.000, C 0.000 }
gfCNCPoint3[1954] = {X 388.0597, Y 53.6000, Z -3.8333, A 0.000, B 0.000, C 0.000 }
gfCNCPoint3[1955] = {X 389.0388, Y 53.7103, Z -3.8333, A 0.000, B 0.000, C 0.000 }
gfCNCPoint3[1956] = {X 389.9688, Y 54.0357, Z -3.8333, A 0.000, B 0.000, C 0.000 }
gfCNCPoint3[1957] = {X 390.8030, Y 54.5599, Z -3.8333, A 0.000, B 0.000, C 0.000 }
gfCNCPoint3[1958] = {X 391.4997, Y 55.2566, Z -3.8333, A 0.000, B 0.000, C 0.000 }
gfCNCPoint3[1959] = {X 392.0239, Y 56.0909, Z -3.8333, A 0.000, B 0.000, C 0.000 }
gfCNCPoint3[1960] = {X 392.3494, Y 57.0209, Z -3.8333, A 0.000, B 0.000, C 0.000 }
gfCNCPoint3[1961] = {X 392.4597, Y 58.0000, Z -3.8333, A 0.000, B 0.000, C 0.000 }
gfCNCPoint3[1962] = {X 392.4595, Y 58.9704, Z -3.8333, A 0.000, B 0.000, C 0.000 }
gfCNCPoint3[1963] = {X 392.3389, Y 59.9578, Z -3.8333, A 0.000, B 0.000, C 0.000 }
gfCNCPoint3[1964] = {X 391.9996, Y 60.8929, Z -3.8333, A 0.000, B 0.000, C 0.000 }
gfCNCPoint3[1965] = {X 391.5562, Y 61.6058, Z -3.8333, A 0.000, B 0.000, C 0.000 }
gfCNCPoint3[1966] = {X 390.9860, Y 62.2220, Z -3.8333, A 0.000, B 0.000, C 0.000 }
gfCNCPoint3[1967] = {X 390.3095, Y 62.7194, Z -3.8333, A 0.000, B 0.000, C 0.000 }
gfCNCPoint3[1968] = {X 389.5513, Y 63.0799, Z -3.8333, A 0.000, B 0.000, C 0.000 }
gfCNCPoint3[1969] = {X 388.7386, Y 63.2907, Z -3.8333, A 0.000, B 0.000, C 0.000 }
gfCNCPoint3[1970] = {X 388.7386, Y 83.9247, Z -3.8333, A 0.000, B 0.000, C 0.000 }
gfCNCPoint3[1971] = {X 388.7366, Y 84.6150, Z -3.8333, A 0.000, B 0.000, C 0.000 }
gfCNCPoint3[1972] = {X 388.6764, Y 86.2799, Z -3.8333, A 0.000, B 0.000, C 0.000 }
gfCNCPoint3[1973] = {X 388.4712, Y 87.9333, Z -3.8333, A 0.000, B 0.000, C 0.000 }
gfCNCPoint3[1974] = {X 388.1226, Y 89.5624, Z -3.8333, A 0.000, B 0.000, C 0.000 }
gfCNCPoint3[1975] = {X 387.5869, Y 91.1606, Z -3.8333, A 0.000, B 0.000, C 0.000 }
gfCNCPoint3[1976] = {X 386.8322, Y 92.6678, Z -3.8333, A 0.000, B 0.000, C 0.000 }
gfCNCPoint3[1977] = {X 385.8736, Y 94.0542, Z -3.8333, A 0.000, B 0.000, C 0.000 }
gfCNCPoint3[1978] = {X 384.7299, Y 95.2924, Z -3.8333, A 0.000, B 0.000, C 0.000 }
gfCNCPoint3[1979] = {X 383.5018, Y 96.3481, Z -3.8333, A 0.000, B 0.000, C 0.000 }
gfCNCPoint3[1980] = {X 382.1870, Y 97.2935, Z -3.8333, A 0.000, B 0.000, C 0.000 }
gfCNCPoint3[1981] = {X 382.4501, Y 97.6950, Z -3.8333, A 0.000, B 0.000, C 0.000 }
gfCNCPoint3[1982] = {X 391.5260, Y 97.6950, Z -3.8333, A 0.000, B 0.000, C 0.000 }
gfCNCPoint3[1983] = {X 391.5260, Y 97.0659, Z -3.8333, A 0.000, B 0.000, C 0.000 }
gfCNCPoint3[1984] = {X 391.6205, Y 96.1101, Z -3.8333, A 0.000, B 0.000, C 0.000 }
gfCNCPoint3[1985] = {X 391.9004, Y 95.1913, Z -3.8333, A 0.000, B 0.000, C 0.000 }
gfCNCPoint3[1986] = {X 392.3549, Y 94.3451, Z -3.8333, A 0.000, B 0.000, C 0.000 }
gfCNCPoint3[1987] = {X 392.9663, Y 93.6043, Z -3.8333, A 0.000, B 0.000, C 0.000 }
gfCNCPoint3[1988] = {X 393.7110, Y 92.9976, Z -3.8333, A 0.000, B 0.000, C 0.000 }
gfCNCPoint3[1989] = {X 394.5600, Y 92.5485, Z -3.8333, A 0.000, B 0.000, C 0.000 }
gfCNCPoint3[1990] = {X 395.4806, Y 92.2745, Z -3.8333, A 0.000, B 0.000, C 0.000 }
gfCNCPoint3[1991] = {X 396.4371, Y 92.1860, Z -3.8333, A 0.000, B 0.000, C 0.000 }
gfCNCPoint3[1992] = {X 397.3327, Y 92.1440, Z -3.8333, A 0.000, B 0.000, C 0.000 }
gfCNCPoint3[1993] = {X 398.2252, Y 92.0588, Z -3.8333, A 0.000, B 0.000, C 0.000 }
gfCNCPoint3[1994] = {X 398.7530, Y 91.9307, Z -3.8333, A 0.000, B 0.000, C 0.000 }
gfCNCPoint3[1995] = {X 399.2389, Y 91.6881, Z -3.8333, A 0.000, B 0.000, C 0.000 }
gfCNCPoint3[1996] = {X 426.8272, Y 74.0194, Z -3.8333, A 0.000, B 0.000, C 0.000 }
gfCNCPoint3[1997] = {X 403.5509, Y 64.8868, Z -3.8333, A 0.000, B 0.000, C 0.000 }
gfCNCPoint3[1998] = {X 401.9167, Y 64.3455, Z -3.8333, A 0.000, B 0.000, C 0.000 }
gfCNCPoint3[1999] = {X 400.2332, Y 63.9864, Z -3.8333, A 0.000, B 0.000, C 0.000 }
gfCNCPoint3[2000] = {X 398.5204, Y 63.8139, Z -3.8333, A 0.000, B 0.000, C 0.000 }
gfCNCPoint3[2001] = {X 397.5547, Y 63.7099, Z -3.8333, A 0.000, B 0.000, C 0.000 }
gfCNCPoint3[2002] = {X 396.6287, Y 63.4166, Z -3.8333, A 0.000, B 0.000, C 0.000 }
gfCNCPoint3[2003] = {X 395.7791, Y 62.9458, Z -3.8333, A 0.000, B 0.000, C 0.000 }
gfCNCPoint3[2004] = {X 395.0396, Y 62.3160, Z -3.8333, A 0.000, B 0.000, C 0.000 }
gfCNCPoint3[2005] = {X 394.4659, Y 61.5933, Z -3.8333, A 0.000, B 0.000, C 0.000 }
gfCNCPoint3[2006] = {X 394.0385, Y 60.7757, Z -3.8333, A 0.000, B 0.000, C 0.000 }
gfCNCPoint3[2007] = {X 393.7727, Y 59.8921, Z -3.8333, A 0.000, B 0.000, C 0.000 }
gfCNCPoint3[2008] = {X 393.6779, Y 58.9744, Z -3.8333, A 0.000, B 0.000, C 0.000 }
gfCNCPoint3[2009] = {X 393.6777, Y 58.0000, Z -3.8333, A 0.000, B 0.000, C 0.000 }
gfCNCPoint3[2010] = {X 393.7668, Y 57.0718, Z -3.8333, A 0.000, B 0.000, C 0.000 }
gfCNCPoint3[2011] = {X 394.0309, Y 56.1774, Z -3.8333, A 0.000, B 0.000, C 0.000 }
gfCNCPoint3[2012] = {X 394.4602, Y 55.3496, Z -3.8333, A 0.000, B 0.000, C 0.000 }
gfCNCPoint3[2013] = {X 395.0391, Y 54.6186, Z -3.8333, A 0.000, B 0.000, C 0.000 }
gfCNCPoint3[2014] = {X 395.7864, Y 53.9833, Z -3.8333, A 0.000, B 0.000, C 0.000 }
gfCNCPoint3[2015] = {X 396.6455, Y 53.5102, Z -3.8333, A 0.000, B 0.000, C 0.000 }
gfCNCPoint3[2016] = {X 397.5819, Y 53.2186, Z -3.8333, A 0.000, B 0.000, C 0.000 }
gfCNCPoint3[2017] = {X 398.5577, Y 53.1200, Z -3.8333, A 0.000, B 0.000, C 0.000 }
gfCNCPoint3[2018] = {X 419.4886, Y 53.1200, Z -3.8333, A 0.000, B 0.000, C 0.000 }
gfCNCPoint3[2019] = {X 420.5534, Y 53.2376, Z -3.8333, A 0.000, B 0.000, C 0.000 }
gfCNCPoint3[2020] = {X 421.5669, Y 53.5847, Z -3.8333, A 0.000, B 0.000, C 0.000 }
gfCNCPoint3[2021] = {X 422.4802, Y 54.1445, Z -3.8333, A 0.000, B 0.000, C 0.000 }
gfCNCPoint3[2022] = {X 423.2494, Y 54.8902, Z -3.8333, A 0.000, B 0.000, C 0.000 }
gfCNCPoint3[2023] = {X 423.8373, Y 55.7857, Z -3.8333, A 0.000, B 0.000, C 0.000 }
gfCNCPoint3[2024] = {X 424.2157, Y 56.7880, Z -3.8333, A 0.000, B 0.000, C 0.000 }
gfCNCPoint3[2025] = {X 424.3663, Y 57.8486, Z -3.8333, A 0.000, B 0.000, C 0.000 }
gfCNCPoint3[2026] = {X 429.8190, Y 59.9735, Z -3.8333, A 0.000, B 0.000, C 0.000 }
gfCNCPoint3[2027] = {X 457.2988, Y 70.8763, Z -3.8333, A 0.000, B 0.000, C 0.000 }
gfCNCPoint3[2028] = {X 457.2993, Y 63.6741, Z -3.8333, A 0.000, B 0.000, C 0.000 }
gfCNCPoint3[2029] = {X 456.2910, Y 63.3058, Z -3.8333, A 0.000, B 0.000, C 0.000 }
gfCNCPoint3[2030] = {X 455.3877, Y 62.7259, Z -3.8333, A 0.000, B 0.000, C 0.000 }
gfCNCPoint3[2031] = {X 454.6330, Y 61.9625, Z -3.8333, A 0.000, B 0.000, C 0.000 }
gfCNCPoint3[2032] = {X 454.0635, Y 61.0527, Z -3.8333, A 0.000, B 0.000, C 0.000 }
gfCNCPoint3[2033] = {X 453.7066, Y 60.0403, Z -3.8333, A 0.000, B 0.000, C 0.000 }
gfCNCPoint3[2034] = {X 453.5798, Y 58.9744, Z -3.8333, A 0.000, B 0.000, C 0.000 }
gfCNCPoint3[2035] = {X 453.5796, Y 58.0000, Z -3.8333, A 0.000, B 0.000, C 0.000 }
gfCNCPoint3[2036] = {X 453.6734, Y 57.0480, Z -3.8333, A 0.000, B 0.000, C 0.000 }
gfCNCPoint3[2037] = {X 453.9511, Y 56.1325, Z -3.8333, A 0.000, B 0.000, C 0.000 }
gfCNCPoint3[2038] = {X 454.4020, Y 55.2888, Z -3.8333, A 0.000, B 0.000, C 0.000 }
gfCNCPoint3[2039] = {X 455.0089, Y 54.5493, Z -3.8333, A 0.000, B 0.000, C 0.000 }
gfCNCPoint3[2040] = {X 455.7484, Y 53.9424, Z -3.8333, A 0.000, B 0.000, C 0.000 }
gfCNCPoint3[2041] = {X 456.5921, Y 53.4915, Z -3.8333, A 0.000, B 0.000, C 0.000 }
gfCNCPoint3[2042] = {X 457.5076, Y 53.2138, Z -3.8333, A 0.000, B 0.000, C 0.000 }
gfCNCPoint3[2043] = {X 458.4596, Y 53.1200, Z -3.8333, A 0.000, B 0.000, C 0.000 }
gfCNCPoint3[2044] = {X 475.0000, Y 53.1200, Z -3.8333, A 0.000, B 0.000, C 0.000 }
gfCNCPoint3[2045] = {X 475.9520, Y 53.2138, Z -3.8333, A 0.000, B 0.000, C 0.000 }
gfCNCPoint3[2046] = {X 476.8675, Y 53.4915, Z -3.8333, A 0.000, B 0.000, C 0.000 }
gfCNCPoint3[2047] = {X 477.7112, Y 53.9424, Z -3.8333, A 0.000, B 0.000, C 0.000 }
gfCNCPoint3[2048] = {X 478.4507, Y 54.5493, Z -3.8333, A 0.000, B 0.000, C 0.000 }
gfCNCPoint3[2049] = {X 479.0576, Y 55.2888, Z -3.8333, A 0.000, B 0.000, C 0.000 }
gfCNCPoint3[2050] = {X 479.5085, Y 56.1325, Z -3.8333, A 0.000, B 0.000, C 0.000 }
gfCNCPoint3[2051] = {X 479.7862, Y 57.0480, Z -3.8333, A 0.000, B 0.000, C 0.000 }
gfCNCPoint3[2052] = {X 479.8800, Y 58.0000, Z -3.8333, A 0.000, B 0.000, C 0.000 }
gfCNCPoint3[2053] = {X 479.8798, Y 58.9744, Z -3.8333, A 0.000, B 0.000, C 0.000 }
gfCNCPoint3[2054] = {X 479.7530, Y 60.0403, Z -3.8333, A 0.000, B 0.000, C 0.000 }
gfCNCPoint3[2055] = {X 479.3961, Y 61.0528, Z -3.8333, A 0.000, B 0.000, C 0.000 }
gfCNCPoint3[2056] = {X 478.8265, Y 61.9627, Z -3.8333, A 0.000, B 0.000, C 0.000 }
gfCNCPoint3[2057] = {X 478.0717, Y 62.7260, Z -3.8333, A 0.000, B 0.000, C 0.000 }
gfCNCPoint3[2058] = {X 477.1683, Y 63.3059, Z -3.8333, A 0.000, B 0.000, C 0.000 }
gfCNCPoint3[2059] = {X 476.1600, Y 63.6742, Z -3.8333, A 0.000, B 0.000, C 0.000 }
gfCNCPoint3[2060] = {X 476.1604, Y 92.3317, Z -3.8333, A 0.000, B 0.000, C 0.000 }
gfCNCPoint3[2061] = {X 476.3634, Y 92.3912, Z -3.8333, A 0.000, B 0.000, C 0.000 }
gfCNCPoint3[2062] = {X 476.5649, Y 92.4557, Z -3.8333, A 0.000, B 0.000, C 0.000 }
gfCNCPoint3[2063] = {X 477.4825, Y 92.8727, Z -3.8333, A 0.000, B 0.000, C 0.000 }
gfCNCPoint3[2064] = {X 478.2942, Y 93.4703, Z -3.8333, A 0.000, B 0.000, C 0.000 }
gfCNCPoint3[2065] = {X 478.9650, Y 94.2225, Z -3.8333, A 0.000, B 0.000, C 0.000 }
gfCNCPoint3[2066] = {X 479.4659, Y 95.0972, Z -3.8333, A 0.000, B 0.000, C 0.000 }
gfCNCPoint3[2067] = {X 479.7753, Y 96.0564, Z -3.8333, A 0.000, B 0.000, C 0.000 }
gfCNCPoint3[2068] = {X 479.8800, Y 97.0589, Z -3.8333, A 0.000, B 0.000, C 0.000 }
gfCNCPoint3[2069] = {X 479.8800, Y 97.6950, Z -3.8333, A 0.000, B 0.000, C 0.000 }
gfCNCPoint3[2070] = {X 479.4000, Y 97.6950, Z -3.8333, A 0.000, B 0.000, C 0.000 }
gfCNCPoint3[2071] = {X 479.4000, Y 98.0000, Z -3.8333, A 0.000, B 0.000, C 0.000 }
gfCNCPoint3[2072] = {X 479.2897, Y 98.9791, Z -3.8333, A 0.000, B 0.000, C 0.000 }
gfCNCPoint3[2073] = {X 478.9643, Y 99.9091, Z -3.8333, A 0.000, B 0.000, C 0.000 }
gfCNCPoint3[2074] = {X 478.4401, Y 100.7434, Z -3.8333, A 0.000, B 0.000, C 0.000 }
gfCNCPoint3[2075] = {X 477.7434, Y 101.4401, Z -3.8333, A 0.000, B 0.000, C 0.000 }
gfCNCPoint3[2076] = {X 476.9091, Y 101.9643, Z -3.8333, A 0.000, B 0.000, C 0.000 }
gfCNCPoint3[2077] = {X 475.9791, Y 102.2897, Z -3.8333, A 0.000, B 0.000, C 0.000 }
gfCNCPoint3[2078] = {X 475.0000, Y 102.4000, Z -3.8333, A 0.000, B 0.000, C 0.000 }
gfCNCPoint3[2079] = {X 458.4596, Y 102.4000, Z -3.8333, A 0.000, B 0.000, C 0.000 }
gfCNCPoint3[2080] = {X 457.4805, Y 102.2897, Z -3.8333, A 0.000, B 0.000, C 0.000 }
gfCNCPoint3[2081] = {X 456.5505, Y 101.9643, Z -3.8333, A 0.000, B 0.000, C 0.000 }
gfCNCPoint3[2082] = {X 455.7162, Y 101.4401, Z -3.8333, A 0.000, B 0.000, C 0.000 }
gfCNCPoint3[2083] = {X 455.0195, Y 100.7434, Z -3.8333, A 0.000, B 0.000, C 0.000 }
gfCNCPoint3[2084] = {X 454.4953, Y 99.9091, Z -3.8333, A 0.000, B 0.000, C 0.000 }
gfCNCPoint3[2085] = {X 454.1699, Y 98.9791, Z -3.8333, A 0.000, B 0.000, C 0.000 }
gfCNCPoint3[2086] = {X 454.0596, Y 98.0000, Z -3.8333, A 0.000, B 0.000, C 0.000 }
gfCNCPoint3[2087] = {X 454.0596, Y 97.0659, Z -3.8333, A 0.000, B 0.000, C 0.000 }
gfCNCPoint3[2088] = {X 454.1492, Y 96.1826, Z -3.8333, A 0.000, B 0.000, C 0.000 }
gfCNCPoint3[2089] = {X 454.4143, Y 95.3353, Z -3.8333, A 0.000, B 0.000, C 0.000 }
gfCNCPoint3[2090] = {X 454.8440, Y 94.5584, Z -3.8333, A 0.000, B 0.000, C 0.000 }
gfCNCPoint3[2091] = {X 455.4210, Y 93.8836, Z -3.8333, A 0.000, B 0.000, C 0.000 }
gfCNCPoint3[2092] = {X 456.1217, Y 93.3384, Z -3.8333, A 0.000, B 0.000, C 0.000 }
gfCNCPoint3[2093] = {X 456.9176, Y 92.9450, Z -3.8333, A 0.000, B 0.000, C 0.000 }
gfCNCPoint3[2094] = {X 457.7763, Y 92.7193, Z -3.8333, A 0.000, B 0.000, C 0.000 }
gfCNCPoint3[2095] = {X 457.7763, Y 85.6495, Z -3.8333, A 0.000, B 0.000, C 0.000 }
gfCNCPoint3[2096] = {X 444.8678, Y 80.5894, Z -3.8333, A 0.000, B 0.000, C 0.000 }
gfCNCPoint3[2097] = {X 420.1035, Y 96.6315, Z -3.8333, A 0.000, B 0.000, C 0.000 }
gfCNCPoint3[2098] = {X 420.1067, Y 97.0659, Z -3.8333, A 0.000, B 0.000, C 0.000 }
gfCNCPoint3[2099] = {X 420.1067, Y 98.0000, Z -3.8333, A 0.000, B 0.000, C 0.000 }
gfCNCPoint3[2100] = {X 419.9964, Y 98.9791, Z -3.8333, A 0.000, B 0.000, C 0.000 }
gfCNCPoint3[2101] = {X 419.6710, Y 99.9091, Z -3.8333, A 0.000, B 0.000, C 0.000 }
gfCNCPoint3[2102] = {X 419.1468, Y 100.7434, Z -3.8333, A 0.000, B 0.000, C 0.000 }
gfCNCPoint3[2103] = {X 418.4501, Y 101.4401, Z -3.8333, A 0.000, B 0.000, C 0.000 }
gfCNCPoint3[2104] = {X 417.6158, Y 101.9643, Z -3.8333, A 0.000, B 0.000, C 0.000 }
gfCNCPoint3[2105] = {X 416.6858, Y 102.2897, Z -3.8333, A 0.000, B 0.000, C 0.000 }
gfCNCPoint3[2106] = {X 415.7067, Y 102.4000, Z -3.8333, A 0.000, B 0.000, C 0.000 }
gfCNCPoint3[2107] = {X 396.4059, Y 102.4000, Z -3.8333, A 0.000, B 0.000, C 0.000 }
gfCNCPoint3[2108] = {X 395.4269, Y 102.2897, Z -3.8333, A 0.000, B 0.000, C 0.000 }
gfCNCPoint3[2109] = {X 394.4969, Y 101.9643, Z -3.8333, A 0.000, B 0.000, C 0.000 }
gfCNCPoint3[2110] = {X 393.6626, Y 101.4401, Z -3.8333, A 0.000, B 0.000, C 0.000 }
gfCNCPoint3[2111] = {X 392.9659, Y 100.7434, Z -3.8333, A 0.000, B 0.000, C 0.000 }
gfCNCPoint3[2112] = {X 392.4417, Y 99.9091, Z -3.8333, A 0.000, B 0.000, C 0.000 }
gfCNCPoint3[2113] = {X 392.1163, Y 98.9791, Z -3.8333, A 0.000, B 0.000, C 0.000 }
gfCNCPoint3[2114] = {X 392.0059, Y 98.0000, Z -3.8333, A 0.000, B 0.000, C 0.000 }
gfCNCPoint3[2115] = {X 392.0059, Y 97.0659, Z -3.8333, A 0.000, B 0.000, C 0.000 }
gfCNCPoint3[2116] = {X 392.1174, Y 96.0820, Z -3.8333, A 0.000, B 0.000, C 0.000 }
gfCNCPoint3[2117] = {X 392.4460, Y 95.1479, Z -3.8333, A 0.000, B 0.000, C 0.000 }
gfCNCPoint3[2118] = {X 392.9752, Y 94.3109, Z -3.8333, A 0.000, B 0.000, C 0.000 }
gfCNCPoint3[2119] = {X 393.6782, Y 93.6135, Z -3.8333, A 0.000, B 0.000, C 0.000 }
gfCNCPoint3[2120] = {X 394.5193, Y 93.0909, Z -3.8333, A 0.000, B 0.000, C 0.000 }
gfCNCPoint3[2121] = {X 395.4560, Y 92.7697, Z -3.8333, A 0.000, B 0.000, C 0.000 }
gfCNCPoint3[2122] = {X 396.4408, Y 92.6661, Z -3.8333, A 0.000, B 0.000, C 0.000 }
gfCNCPoint3[2123] = {X 397.3639, Y 92.6230, Z -3.8333, A 0.000, B 0.000, C 0.000 }
gfCNCPoint3[2124] = {X 398.2839, Y 92.5352, Z -3.8333, A 0.000, B 0.000, C 0.000 }
gfCNCPoint3[2125] = {X 398.9176, Y 92.3816, Z -3.8333, A 0.000, B 0.000, C 0.000 }
gfCNCPoint3[2126] = {X 399.5010, Y 92.0903, Z -3.8333, A 0.000, B 0.000, C 0.000 }
gfCNCPoint3[2127] = {X 405.1771, Y 88.4328, Z -3.8333, A 0.000, B 0.000, C 0.000 }
gfCNCPoint3[2128] = {X 427.8791, Y 73.9165, Z -3.8333, A 0.000, B 0.000, C 0.000 }
gfCNCPoint3[2129] = {X 403.7262, Y 64.4399, Z -3.8333, A 0.000, B 0.000, C 0.000 }
gfCNCPoint3[2130] = {X 402.0392, Y 63.8813, Z -3.8333, A 0.000, B 0.000, C 0.000 }
gfCNCPoint3[2131] = {X 400.3011, Y 63.5112, Z -3.8333, A 0.000, B 0.000, C 0.000 }
gfCNCPoint3[2132] = {X 398.5328, Y 63.3340, Z -3.8333, A 0.000, B 0.000, C 0.000 }
gfCNCPoint3[2133] = {X 397.5578, Y 63.2190, Z -3.8333, A 0.000, B 0.000, C 0.000 }
gfCNCPoint3[2134] = {X 396.6326, Y 62.8906, Z -3.8333, A 0.000, B 0.000, C 0.000 }
gfCNCPoint3[2135] = {X 395.8033, Y 62.3652, Z -3.8333, A 0.000, B 0.000, C 0.000 }
gfCNCPoint3[2136] = {X 395.1110, Y 61.6691, Z -3.8333, A 0.000, B 0.000, C 0.000 }
gfCNCPoint3[2137] = {X 394.5904, Y 60.8367, Z -3.8333, A 0.000, B 0.000, C 0.000 }
gfCNCPoint3[2138] = {X 394.2672, Y 59.9097, Z -3.8333, A 0.000, B 0.000, C 0.000 }
gfCNCPoint3[2139] = {X 394.1577, Y 58.9340, Z -3.8333, A 0.000, B 0.000, C 0.000 }
gfCNCPoint3[2140] = {X 394.1577, Y 58.0000, Z -3.8333, A 0.000, B 0.000, C 0.000 }
gfCNCPoint3[2141] = {X 394.2680, Y 57.0209, Z -3.8333, A 0.000, B 0.000, C 0.000 }
gfCNCPoint3[2142] = {X 394.5935, Y 56.0909, Z -3.8333, A 0.000, B 0.000, C 0.000 }
gfCNCPoint3[2143] = {X 395.1177, Y 55.2566, Z -3.8333, A 0.000, B 0.000, C 0.000 }
gfCNCPoint3[2144] = {X 395.8144, Y 54.5599, Z -3.8333, A 0.000, B 0.000, C 0.000 }
gfCNCPoint3[2145] = {X 396.6486, Y 54.0357, Z -3.8333, A 0.000, B 0.000, C 0.000 }
gfCNCPoint3[2146] = {X 397.5786, Y 53.7103, Z -3.8333, A 0.000, B 0.000, C 0.000 }
gfCNCPoint3[2147] = {X 398.5577, Y 53.6000, Z -3.8333, A 0.000, B 0.000, C 0.000 }
gfCNCPoint3[2148] = {X 419.4886, Y 53.6000, Z -3.8333, A 0.000, B 0.000, C 0.000 }
gfCNCPoint3[2149] = {X 420.4677, Y 53.7103, Z -3.8333, A 0.000, B 0.000, C 0.000 }
gfCNCPoint3[2150] = {X 421.3977, Y 54.0357, Z -3.8333, A 0.000, B 0.000, C 0.000 }
gfCNCPoint3[2151] = {X 422.2320, Y 54.5599, Z -3.8333, A 0.000, B 0.000, C 0.000 }
gfCNCPoint3[2152] = {X 422.9287, Y 55.2566, Z -3.8333, A 0.000, B 0.000, C 0.000 }
gfCNCPoint3[2153] = {X 423.4529, Y 56.0909, Z -3.8333, A 0.000, B 0.000, C 0.000 }
gfCNCPoint3[2154] = {X 423.7783, Y 57.0209, Z -3.8333, A 0.000, B 0.000, C 0.000 }
gfCNCPoint3[2155] = {X 423.8886, Y 58.0000, Z -3.8333, A 0.000, B 0.000, C 0.000 }
gfCNCPoint3[2156] = {X 423.8886, Y 58.1776, Z -3.8333, A 0.000, B 0.000, C 0.000 }
gfCNCPoint3[2157] = {X 429.6420, Y 60.4197, Z -3.8333, A 0.000, B 0.000, C 0.000 }
gfCNCPoint3[2158] = {X 457.7787, Y 71.5831, Z -3.8333, A 0.000, B 0.000, C 0.000 }
gfCNCPoint3[2159] = {X 457.7793, Y 63.2812, Z -3.8333, A 0.000, B 0.000, C 0.000 }
gfCNCPoint3[2160] = {X 456.9201, Y 63.0559, Z -3.8333, A 0.000, B 0.000, C 0.000 }
gfCNCPoint3[2161] = {X 456.1236, Y 62.6627, Z -3.8333, A 0.000, B 0.000, C 0.000 }
gfCNCPoint3[2162] = {X 455.4223, Y 62.1176, Z -3.8333, A 0.000, B 0.000, C 0.000 }
gfCNCPoint3[2163] = {X 454.8448, Y 61.4426, Z -3.8333, A 0.000, B 0.000, C 0.000 }
gfCNCPoint3[2164] = {X 454.4146, Y 60.6655, Z -3.8333, A 0.000, B 0.000, C 0.000 }
gfCNCPoint3[2165] = {X 454.1493, Y 59.8178, Z -3.8333, A 0.000, B 0.000, C 0.000 }
gfCNCPoint3[2166] = {X 454.0596, Y 58.9340, Z -3.8333, A 0.000, B 0.000, C 0.000 }
gfCNCPoint3[2167] = {X 454.0596, Y 58.0000, Z -3.8333, A 0.000, B 0.000, C 0.000 }
gfCNCPoint3[2168] = {X 454.1699, Y 57.0209, Z -3.8333, A 0.000, B 0.000, C 0.000 }
gfCNCPoint3[2169] = {X 454.4953, Y 56.0909, Z -3.8333, A 0.000, B 0.000, C 0.000 }
gfCNCPoint3[2170] = {X 455.0195, Y 55.2566, Z -3.8333, A 0.000, B 0.000, C 0.000 }
gfCNCPoint3[2171] = {X 455.7162, Y 54.5599, Z -3.8333, A 0.000, B 0.000, C 0.000 }
gfCNCPoint3[2172] = {X 456.5505, Y 54.0357, Z -3.8333, A 0.000, B 0.000, C 0.000 }
gfCNCPoint3[2173] = {X 457.4805, Y 53.7103, Z -3.8333, A 0.000, B 0.000, C 0.000 }
gfCNCPoint3[2174] = {X 458.4596, Y 53.6000, Z -3.8333, A 0.000, B 0.000, C 0.000 }
gfCNCPoint3[2175] = {X 475.0000, Y 53.6000, Z -3.8333, A 0.000, B 0.000, C 0.000 }
gfCNCPoint3[2176] = {X 475.9791, Y 53.7103, Z -3.8333, A 0.000, B 0.000, C 0.000 }
gfCNCPoint3[2177] = {X 476.9091, Y 54.0357, Z -3.8333, A 0.000, B 0.000, C 0.000 }
gfCNCPoint3[2178] = {X 477.7434, Y 54.5599, Z -3.8333, A 0.000, B 0.000, C 0.000 }
gfCNCPoint3[2179] = {X 478.4401, Y 55.2566, Z -3.8333, A 0.000, B 0.000, C 0.000 }
gfCNCPoint3[2180] = {X 478.9643, Y 56.0909, Z -3.8333, A 0.000, B 0.000, C 0.000 }
gfCNCPoint3[2181] = {X 479.2897, Y 57.0209, Z -3.8333, A 0.000, B 0.000, C 0.000 }
gfCNCPoint3[2182] = {X 479.4000, Y 58.0000, Z -3.8333, A 0.000, B 0.000, C 0.000 }
gfCNCPoint3[2183] = {X 479.3998, Y 58.9704, Z -3.8333, A 0.000, B 0.000, C 0.000 }
gfCNCPoint3[2184] = {X 479.3040, Y 59.8483, Z -3.8333, A 0.000, B 0.000, C 0.000 }
gfCNCPoint3[2185] = {X 479.0347, Y 60.6894, Z -3.8333, A 0.000, B 0.000, C 0.000 }
gfCNCPoint3[2186] = {X 478.6029, Y 61.4598, Z -3.8333, A 0.000, B 0.000, C 0.000 }
gfCNCPoint3[2187] = {X 478.0259, Y 62.1284, Z -3.8333, A 0.000, B 0.000, C 0.000 }
gfCNCPoint3[2188] = {X 477.3270, Y 62.6684, Z -3.8333, A 0.000, B 0.000, C 0.000 }
gfCNCPoint3[2189] = {X 476.5344, Y 63.0578, Z -3.8333, A 0.000, B 0.000, C 0.000 }
gfCNCPoint3[2190] = {X 475.6800, Y 63.2812, Z -3.8333, A 0.000, B 0.000, C 0.000 }
gfCNCPoint3[2191] = {X 475.6804, Y 92.7045, Z -3.8333, A 0.000, B 0.000, C 0.000 }
gfCNCPoint3[2192] = {X 476.0490, Y 92.7990, Z -3.8333, A 0.000, B 0.000, C 0.000 }
gfCNCPoint3[2193] = {X 476.4127, Y 92.9110, Z -3.8333, A 0.000, B 0.000, C 0.000 }
gfCNCPoint3[2194] = {X 477.2396, Y 93.2867, Z -3.8333, A 0.000, B 0.000, C 0.000 }
gfCNCPoint3[2195] = {X 477.9710, Y 93.8252, Z -3.8333, A 0.000, B 0.000, C 0.000 }
gfCNCPoint3[2196] = {X 478.5755, Y 94.5031, Z -3.8333, A 0.000, B 0.000, C 0.000 }
gfCNCPoint3[2197] = {X 479.0268, Y 95.2912, Z -3.8333, A 0.000, B 0.000, C 0.000 }
gfCNCPoint3[2198] = {X 479.3057, Y 96.1555, Z -3.8333, A 0.000, B 0.000, C 0.000 }
gfCNCPoint3[2199] = {X 479.4000, Y 97.0589, Z -3.8333, A 0.000, B 0.000, C 0.000 }
gfCNCPoint3[2200] = {X 479.4000, Y 97.6950, Z -3.8333, A 0.000, B 0.000, C 0.000 }
gfCNCPoint3[2201] = {X 479.8800, Y 97.6950, Z -3.8333, A 0.000, B 0.000, C 0.000 }
gfCNCPoint3[2202] = {X 507.6816, Y 97.6950, Z -3.8333, A 0.000, B 0.000, C 0.000 }
gfCNCPoint3[2203] = {X 507.6816, Y 100.0950, Z -3.8333, A 0.000, B 0.000, C 0.000 }
gfCNCPoint3[2204] = {X 600.0148, Y 100.0950, Z -3.8333, A 0.000, B 0.000, C 0.000 }
gfCNCPoint3[2205] = {X 600.0672, Y 100.0698, Z -3.8333, A 0.000, B 0.000, C 0.000 }
gfCNCPoint3[2206] = {X 600.0948, Y 100.0187, Z -3.8333, A 0.000, B 0.000, C 0.000 }
gfCNCPoint3[2207] = {X 600.0965, Y 99.1431, Z -3.8333, A 0.000, B 0.000, C 0.000 }
gfCNCPoint3[2208] = {X 600.0965, Y 49.8790, Z -3.8333, A 0.000, B 0.000, C 0.000 }
gfCNCPoint3[2209] = {X 601.1111, Y 49.7518, Z -3.8333, A 0.000, B 0.000, C 0.000 }
gfCNCPoint3[2210] = {X 602.0769, Y 49.4160, Z -3.8333, A 0.000, B 0.000, C 0.000 }
gfCNCPoint3[2211] = {X 602.9515, Y 48.8862, Z -3.8333, A 0.000, B 0.000, C 0.000 }
gfCNCPoint3[2212] = {X 603.6965, Y 48.1859, Z -3.8333, A 0.000, B 0.000, C 0.000 }
gfCNCPoint3[2213] = {X 603.6965, Y 47.3865, Z -3.8333, A 0.000, B 0.000, C 0.000 }
gfCNCPoint3[2214] = {X 603.1503, Y 48.0718, Z -3.8333, A 0.000, B 0.000, C 0.000 }
gfCNCPoint3[2215] = {X 602.4790, Y 48.6352, Z -3.8333, A 0.000, B 0.000, C 0.000 }
gfCNCPoint3[2216] = {X 601.7094, Y 49.0544, Z -3.8333, A 0.000, B 0.000, C 0.000 }
gfCNCPoint3[2217] = {X 600.8720, Y 49.3127, Z -3.8333, A 0.000, B 0.000, C 0.000 }
gfCNCPoint3[2218] = {X 600.0000, Y 49.4000, Z -3.8333, A 0.000, B 0.000, C 0.000 }
gfCNCPoint3[2219] = {X 593.5565, Y 49.4000, Z -3.8333, A 0.000, B 0.000, C 0.000 }
gfCNCPoint3[2220] = {X 592.5988, Y 49.2945, Z -3.8333, A 0.000, B 0.000, C 0.000 }
gfCNCPoint3[2221] = {X 591.6870, Y 48.9831, Z -3.8333, A 0.000, B 0.000, C 0.000 }
gfCNCPoint3[2222] = {X 590.8648, Y 48.4806, Z -3.8333, A 0.000, B 0.000, C 0.000 }
gfCNCPoint3[2223] = {X 590.1717, Y 47.8112, Z -3.8333, A 0.000, B 0.000, C 0.000 }
gfCNCPoint3[2224] = {X 589.6410, Y 47.0071, Z -3.8333, A 0.000, B 0.000, C 0.000 }
gfCNCPoint3[2225] = {X 589.3741, Y 46.3664, Z -3.8333, A 0.000, B 0.000, C 0.000 }
gfCNCPoint3[2226] = {X 589.2113, Y 45.6918, Z -3.8333, A 0.000, B 0.000, C 0.000 }
gfCNCPoint3[2227] = {X 589.1565, Y 45.0000, Z -3.8333, A 0.000, B 0.000, C 0.000 }
gfCNCPoint3[2228] = {X 589.1565, Y 44.0641, Z -3.8333, A 0.000, B 0.000, C 0.000 }
gfCNCPoint3[2229] = {X 589.2610, Y 43.1277, Z -3.8333, A 0.000, B 0.000, C 0.000 }
gfCNCPoint3[2230] = {X 589.5605, Y 42.2345, Z -3.8333, A 0.000, B 0.000, C 0.000 }
gfCNCPoint3[2231] = {X 590.0417, Y 41.4245, Z -3.8333, A 0.000, B 0.000, C 0.000 }
gfCNCPoint3[2232] = {X 590.6830, Y 40.7343, Z -3.8333, A 0.000, B 0.000, C 0.000 }
gfCNCPoint3[2233] = {X 590.6844, Y 40.3069, Z -3.8333, A 0.000, B 0.000, C 0.000 }
gfCNCPoint3[2234] = {X 590.6835, Y 35.2175, Z -3.8333, A 0.000, B 0.000, C 0.000 }
gfCNCPoint3[2235] = {X 590.6833, Y 33.9400, Z -3.8333, A 0.000, B 0.000, C 0.000 }
gfCNCPoint3[2236] = {X 585.5192, Y 46.6830, Z -3.8333, A 0.000, B 0.000, C 0.000 }
gfCNCPoint3[2237] = {X 585.4476, Y 46.8466, Z -3.8333, A 0.000, B 0.000, C 0.000 }
gfCNCPoint3[2238] = {X 585.3694, Y 47.0071, Z -3.8333, A 0.000, B 0.000, C 0.000 }
gfCNCPoint3[2239] = {X 585.1701, Y 47.3558, Z -3.8333, A 0.000, B 0.000, C 0.000 }
gfCNCPoint3[2240] = {X 584.9398, Y 47.6848, Z -3.8333, A 0.000, B 0.000, C 0.000 }
gfCNCPoint3[2241] = {X 584.4757, Y 48.1982, Z -3.8333, A 0.000, B 0.000, C 0.000 }
gfCNCPoint3[2242] = {X 583.9368, Y 48.6325, Z -3.8333, A 0.000, B 0.000, C 0.000 }
gfCNCPoint3[2243] = {X 583.3365, Y 48.9769, Z -3.8333, A 0.000, B 0.000, C 0.000 }
gfCNCPoint3[2244] = {X 582.4111, Y 49.2946, Z -3.8333, A 0.000, B 0.000, C 0.000 }
gfCNCPoint3[2245] = {X 581.4384, Y 49.4000, Z -3.8333, A 0.000, B 0.000, C 0.000 }
gfCNCPoint3[2246] = {X 580.4664, Y 49.2878, Z -3.8333, A 0.000, B 0.000, C 0.000 }
gfCNCPoint3[2247] = {X 579.5433, Y 48.9635, Z -3.8333, A 0.000, B 0.000, C 0.000 }
gfCNCPoint3[2248] = {X 578.7146, Y 48.4433, Z -3.8333, A 0.000, B 0.000, C 0.000 }
gfCNCPoint3[2249] = {X 578.0214, Y 47.7529, Z -3.8333, A 0.000, B 0.000, C 0.000 }
gfCNCPoint3[2250] = {X 577.4979, Y 46.9263, Z -3.8333, A 0.000, B 0.000, C 0.000 }
gfCNCPoint3[2251] = {X 577.4375, Y 46.7968, Z -3.8333, A 0.000, B 0.000, C 0.000 }
gfCNCPoint3[2252] = {X 577.3813, Y 46.6655, Z -3.8333, A 0.000, B 0.000, C 0.000 }
gfCNCPoint3[2253] = {X 572.0986, Y 33.7478, Z -3.8333, A 0.000, B 0.000, C 0.000 }
gfCNCPoint3[2254] = {X 572.0989, Y 40.7329, Z -3.8333, A 0.000, B 0.000, C 0.000 }
gfCNCPoint3[2255] = {X 572.7435, Y 41.4221, Z -3.8333, A 0.000, B 0.000, C 0.000 }
gfCNCPoint3[2256] = {X 573.2264, Y 42.2328, Z -3.8333, A 0.000, B 0.000, C 0.000 }
gfCNCPoint3[2257] = {X 573.5253, Y 43.1278, Z -3.8333, A 0.000, B 0.000, C 0.000 }
gfCNCPoint3[2258] = {X 573.6264, Y 44.0660, Z -3.8333, A 0.000, B 0.000, C 0.000 }
gfCNCPoint3[2259] = {X 573.6264, Y 45.0000, Z -3.8333, A 0.000, B 0.000, C 0.000 }
gfCNCPoint3[2260] = {X 573.5140, Y 45.9884, Z -3.8333, A 0.000, B 0.000, C 0.000 }
gfCNCPoint3[2261] = {X 573.1824, Y 46.9263, Z -3.8333, A 0.000, B 0.000, C 0.000 }
gfCNCPoint3[2262] = {X 572.6569, Y 47.7553, Z -3.8333, A 0.000, B 0.000, C 0.000 }
gfCNCPoint3[2263] = {X 571.9608, Y 48.4472, Z -3.8333, A 0.000, B 0.000, C 0.000 }
gfCNCPoint3[2264] = {X 571.1286, Y 48.9676, Z -3.8333, A 0.000, B 0.000, C 0.000 }
gfCNCPoint3[2265] = {X 570.2018, Y 49.2905, Z -3.8333, A 0.000, B 0.000, C 0.000 }
gfCNCPoint3[2266] = {X 569.2264, Y 49.4000, Z -3.8333, A 0.000, B 0.000, C 0.000 }
gfCNCPoint3[2267] = {X 562.4443, Y 49.4000, Z -3.8333, A 0.000, B 0.000, C 0.000 }
gfCNCPoint3[2268] = {X 561.4652, Y 49.2897, Z -3.8333, A 0.000, B 0.000, C 0.000 }
gfCNCPoint3[2269] = {X 560.5352, Y 48.9643, Z -3.8333, A 0.000, B 0.000, C 0.000 }
gfCNCPoint3[2270] = {X 559.7009, Y 48.4401, Z -3.8333, A 0.000, B 0.000, C 0.000 }
gfCNCPoint3[2271] = {X 559.0042, Y 47.7434, Z -3.8333, A 0.000, B 0.000, C 0.000 }
gfCNCPoint3[2272] = {X 558.4800, Y 46.9091, Z -3.8333, A 0.000, B 0.000, C 0.000 }
gfCNCPoint3[2273] = {X 558.1546, Y 45.9791, Z -3.8333, A 0.000, B 0.000, C 0.000 }
gfCNCPoint3[2274] = {X 558.0443, Y 45.0000, Z -3.8333, A 0.000, B 0.000, C 0.000 }
gfCNCPoint3[2275] = {X 558.0443, Y 44.0643, Z -3.8333, A 0.000, B 0.000, C 0.000 }
gfCNCPoint3[2276] = {X 558.1485, Y 43.1276, Z -3.8333, A 0.000, B 0.000, C 0.000 }
gfCNCPoint3[2277] = {X 558.4483, Y 42.2342, Z -3.8333, A 0.000, B 0.000, C 0.000 }
gfCNCPoint3[2278] = {X 558.9300, Y 41.4242, Z -3.8333, A 0.000, B 0.000, C 0.000 }
gfCNCPoint3[2279] = {X 559.5721, Y 40.7343, Z -3.8333, A 0.000, B 0.000, C 0.000 }
gfCNCPoint3[2280] = {X 559.5721, Y 9.2673, Z -3.8333, A 0.000, B 0.000, C 0.000 }
gfCNCPoint3[2281] = {X 558.9274, Y 8.5781, Z -3.8333, A 0.000, B 0.000, C 0.000 }
gfCNCPoint3[2282] = {X 558.4444, Y 7.7673, Z -3.8333, A 0.000, B 0.000, C 0.000 }
gfCNCPoint3[2283] = {X 558.1455, Y 6.8722, Z -3.8333, A 0.000, B 0.000, C 0.000 }
gfCNCPoint3[2284] = {X 558.0443, Y 5.9339, Z -3.8333, A 0.000, B 0.000, C 0.000 }
gfCNCPoint3[2285] = {X 558.0443, Y 5.0000, Z -3.8333, A 0.000, B 0.000, C 0.000 }
gfCNCPoint3[2286] = {X 558.1353, Y 4.1097, Z -3.8333, A 0.000, B 0.000, C 0.000 }
gfCNCPoint3[2287] = {X 558.4046, Y 3.2562, Z -3.8333, A 0.000, B 0.000, C 0.000 }
gfCNCPoint3[2288] = {X 558.9155, Y 2.3718, Z -3.8333, A 0.000, B 0.000, C 0.000 }
gfCNCPoint3[2289] = {X 559.6166, Y 1.6290, Z -3.8333, A 0.000, B 0.000, C 0.000 }
gfCNCPoint3[2290] = {X 560.4700, Y 1.0678, Z -3.8333, A 0.000, B 0.000, C 0.000 }
gfCNCPoint3[2291] = {X 561.4298, Y 0.7185, Z -3.8333, A 0.000, B 0.000, C 0.000 }
gfCNCPoint3[2292] = {X 562.4443, Y 0.6000, Z -3.8333, A 0.000, B 0.000, C 0.000 }
gfCNCPoint3[2293] = {X 570.9376, Y 0.6000, Z -3.8333, A 0.000, B 0.000, C 0.000 }
gfCNCPoint3[2294] = {X 571.9520, Y 0.7185, Z -3.8333, A 0.000, B 0.000, C 0.000 }
gfCNCPoint3[2295] = {X 572.9119, Y 1.0678, Z -3.8333, A 0.000, B 0.000, C 0.000 }
gfCNCPoint3[2296] = {X 573.7653, Y 1.6290, Z -3.8333, A 0.000, B 0.000, C 0.000 }
gfCNCPoint3[2297] = {X 574.4663, Y 2.3718, Z -3.8333, A 0.000, B 0.000, C 0.000 }
gfCNCPoint3[2298] = {X 574.9772, Y 3.2562, Z -3.8333, A 0.000, B 0.000, C 0.000 }
gfCNCPoint3[2299] = {X 575.2317, Y 4.0407, Z -3.8333, A 0.000, B 0.000, C 0.000 }
gfCNCPoint3[2300] = {X 575.3353, Y 4.8589, Z -3.8333, A 0.000, B 0.000, C 0.000 }
gfCNCPoint3[2301] = {X 580.1328, Y 4.7050, Z -3.8333, A 0.000, B 0.000, C 0.000 }
gfCNCPoint3[2302] = {X 580.1364, Y 4.8525, Z -3.8333, A 0.000, B 0.000, C 0.000 }
gfCNCPoint3[2303] = {X 580.1376, Y 5.0000, Z -3.8333, A 0.000, B 0.000, C 0.000 }
gfCNCPoint3[2304] = {X 580.1368, Y 6.0531, Z -3.8333, A 0.000, B 0.000, C 0.000 }
gfCNCPoint3[2305] = {X 580.0609, Y 7.1194, Z -3.8333, A 0.000, B 0.000, C 0.000 }
gfCNCPoint3[2306] = {X 579.8618, Y 8.1697, Z -3.8333, A 0.000, B 0.000, C 0.000 }
gfCNCPoint3[2307] = {X 581.1999, Y 11.4542, Z -3.8333, A 0.000, B 0.000, C 0.000 }
gfCNCPoint3[2308] = {X 582.6184, Y 7.9848, Z -3.8333, A 0.000, B 0.000, C 0.000 }
gfCNCPoint3[2309] = {X 582.4489, Y 6.9996, Z -3.8333, A 0.000, B 0.000, C 0.000 }
gfCNCPoint3[2310] = {X 582.3872, Y 6.0018, Z -3.8333, A 0.000, B 0.000, C 0.000 }
gfCNCPoint3[2311] = {X 582.3870, Y 5.0000, Z -3.8333, A 0.000, B 0.000, C 0.000 }
gfCNCPoint3[2312] = {X 582.3881, Y 4.8525, Z -3.8333, A 0.000, B 0.000, C 0.000 }
gfCNCPoint3[2313] = {X 582.3917, Y 4.7050, Z -3.8333, A 0.000, B 0.000, C 0.000 }
gfCNCPoint3[2314] = {X 580.1328, Y 4.7050, Z -3.8333, A 0.000, B 0.000, C 0.000 }
gfCNCPoint3[2315] = {X 577.7341, Y 4.7820, Z -3.8333, A 0.000, B 0.000, C 0.000 }
gfCNCPoint3[2316] = {X 577.7367, Y 4.8910, Z -3.8333, A 0.000, B 0.000, C 0.000 }
gfCNCPoint3[2317] = {X 577.7376, Y 5.0000, Z -3.8333, A 0.000, B 0.000, C 0.000 }
gfCNCPoint3[2318] = {X 577.7370, Y 6.0220, Z -3.8333, A 0.000, B 0.000, C 0.000 }
gfCNCPoint3[2319] = {X 577.6239, Y 7.1720, Z -3.8333, A 0.000, B 0.000, C 0.000 }
gfCNCPoint3[2320] = {X 577.3178, Y 8.2863, Z -3.8333, A 0.000, B 0.000, C 0.000 }
gfCNCPoint3[2321] = {X 581.1958, Y 17.8055, Z -3.8333, A 0.000, B 0.000, C 0.000 }
gfCNCPoint3[2322] = {X 585.1516, Y 8.1309, Z -3.8333, A 0.000, B 0.000, C 0.000 }
gfCNCPoint3[2323] = {X 584.8835, Y 7.0758, Z -3.8333, A 0.000, B 0.000, C 0.000 }
gfCNCPoint3[2324] = {X 584.7872, Y 5.9914, Z -3.8333, A 0.000, B 0.000, C 0.000 }
gfCNCPoint3[2325] = {X 584.7870, Y 5.0000, Z -3.8333, A 0.000, B 0.000, C 0.000 }
gfCNCPoint3[2326] = {X 584.7878, Y 4.8910, Z -3.8333, A 0.000, B 0.000, C 0.000 }
gfCNCPoint3[2327] = {X 584.7905, Y 4.7820, Z -3.8333, A 0.000, B 0.000, C 0.000 }
gfCNCPoint3[2328] = {X 584.9505, Y 3.5174, Z -3.8333, A 0.000, B 0.000, C 0.000 }
gfCNCPoint3[2329] = {X 585.3438, Y 2.3050, Z -3.8333, A 0.000, B 0.000, C 0.000 }
gfCNCPoint3[2330] = {X 577.1807, Y 2.3050, Z -3.8333, A 0.000, B 0.000, C 0.000 }
gfCNCPoint3[2331] = {X 577.5740, Y 3.5174, Z -3.8333, A 0.000, B 0.000, C 0.000 }
gfCNCPoint3[2332] = {X 577.7341, Y 4.7820, Z -3.8333, A 0.000, B 0.000, C 0.000 }
gfCNCPoint3[2333] = {X 575.3353, Y 4.8589, Z -3.8333, A 0.000, B 0.000, C 0.000 }
gfCNCPoint3[2334] = {X 575.3370, Y 4.9294, Z -3.8333, A 0.000, B 0.000, C 0.000 }
gfCNCPoint3[2335] = {X 575.3376, Y 5.0000, Z -3.8333, A 0.000, B 0.000, C 0.000 }
gfCNCPoint3[2336] = {X 575.3372, Y 5.9910, Z -3.8333, A 0.000, B 0.000, C 0.000 }
gfCNCPoint3[2337] = {X 575.2576, Y 6.7689, Z -3.8333, A 0.000, B 0.000, C 0.000 }
gfCNCPoint3[2338] = {X 575.0416, Y 7.5204, Z -3.8333, A 0.000, B 0.000, C 0.000 }
gfCNCPoint3[2339] = {X 574.6960, Y 8.2218, Z -3.8333, A 0.000, B 0.000, C 0.000 }
gfCNCPoint3[2340] = {X 575.2866, Y 9.6573, Z -3.8333, A 0.000, B 0.000, C 0.000 }
gfCNCPoint3[2341] = {X 581.1912, Y 24.1581, Z -3.8333, A 0.000, B 0.000, C 0.000 }
gfCNCPoint3[2342] = {X 587.7570, Y 8.1001, Z -3.8333, A 0.000, B 0.000, C 0.000 }
gfCNCPoint3[2343] = {X 587.4434, Y 7.4144, Z -3.8333, A 0.000, B 0.000, C 0.000 }
gfCNCPoint3[2344] = {X 587.2515, Y 6.6852, Z -3.8333, A 0.000, B 0.000, C 0.000 }
gfCNCPoint3[2345] = {X 587.1870, Y 5.9340, Z -3.8333, A 0.000, B 0.000, C 0.000 }
gfCNCPoint3[2346] = {X 587.1870, Y 5.0000, Z -3.8333, A 0.000, B 0.000, C 0.000 }
gfCNCPoint3[2347] = {X 587.2780, Y 4.1097, Z -3.8333, A 0.000, B 0.000, C 0.000 }
gfCNCPoint3[2348] = {X 587.5473, Y 3.2562, Z -3.8333, A 0.000, B 0.000, C 0.000 }
gfCNCPoint3[2349] = {X 588.0582, Y 2.3718, Z -3.8333, A 0.000, B 0.000, C 0.000 }
gfCNCPoint3[2350] = {X 588.7592, Y 1.6290, Z -3.8333, A 0.000, B 0.000, C 0.000 }
gfCNCPoint3[2351] = {X 589.6127, Y 1.0678, Z -3.8333, A 0.000, B 0.000, C 0.000 }
gfCNCPoint3[2352] = {X 590.5725, Y 0.7185, Z -3.8333, A 0.000, B 0.000, C 0.000 }
gfCNCPoint3[2353] = {X 591.5870, Y 0.6000, Z -3.8333, A 0.000, B 0.000, C 0.000 }
gfCNCPoint3[2354] = {X 600.0000, Y 0.6000, Z -3.8333, A 0.000, B 0.000, C 0.000 }
gfCNCPoint3[2355] = {X 600.8720, Y 0.6873, Z -3.8333, A 0.000, B 0.000, C 0.000 }
gfCNCPoint3[2356] = {X 601.7094, Y 0.9456, Z -3.8333, A 0.000, B 0.000, C 0.000 }
gfCNCPoint3[2357] = {X 602.4790, Y 1.3648, Z -3.8333, A 0.000, B 0.000, C 0.000 }
gfCNCPoint3[2358] = {X 603.1503, Y 1.9282, Z -3.8333, A 0.000, B 0.000, C 0.000 }
gfCNCPoint3[2359] = {X 603.6965, Y 2.6135, Z -3.8333, A 0.000, B 0.000, C 0.000 }
gfCNCPoint3[2360] = {X 603.6965, Y 1.8141, Z -3.8333, A 0.000, B 0.000, C 0.000 }
gfCNCPoint3[2361] = {X 602.9512, Y 1.1135, Z -3.8333, A 0.000, B 0.000, C 0.000 }
gfCNCPoint3[2362] = {X 602.0763, Y 0.5837, Z -3.8333, A 0.000, B 0.000, C 0.000 }
gfCNCPoint3[2363] = {X 601.1101, Y 0.2479, Z -3.8333, A 0.000, B 0.000, C 0.000 }
gfCNCPoint3[2364] = {X 600.0951, Y 0.1209, Z -3.8333, A 0.000, B 0.000, C 0.000 }
gfCNCPoint3[2365] = {X 600.0948, Y -0.0187, Z -3.8333, A 0.000, B 0.000, C 0.000 }
gfCNCPoint3[2366] = {X 600.0672, Y -0.0698, Z -3.8333, A 0.000, B 0.000, C 0.000 }
gfCNCPoint3[2367] = {X 600.0148, Y -0.0950, Z -3.8333, A 0.000, B 0.000, C 0.000 }
gfCNCPoint3[2368] = {X 351.5650, Y -0.0950, Z -3.8333, A 0.000, B 0.000, C 0.000 }
gfCNCPoint3[2369] = {X 351.4055, Y -0.1247, Z -3.8333, A 0.000, B 0.000, C 0.000 }
gfCNCPoint3[2370] = {X 348.9096, Y -0.4711, Z -3.8333, A 0.000, B 0.000, C 0.000 }
gfCNCPoint3[2371] = {X 346.3922, Y -0.5819, Z -3.8333, A 0.000, B 0.000, C 0.000 }
gfCNCPoint3[2372] = {X 343.8755, Y -0.4562, Z -3.8333, A 0.000, B 0.000, C 0.000 }
gfCNCPoint3[2373] = {X 341.3817, Y -0.0950, Z -3.8333, A 0.000, B 0.000, C 0.000 }
gfCNCPoint3[2374] = {X -0.0148, Y -0.0950, Z -3.8333, A 0.000, B 0.000, C 0.000 }
gfCNCPoint3[2375] = {X -0.0672, Y -0.0698, Z -3.8333, A 0.000, B 0.000, C 0.000 }
gfCNCPoint3[2376] = {X -0.0948, Y -0.0187, Z -3.8333, A 0.000, B 0.000, C 0.000 }
gfCNCPoint3[2377] = {X -0.0965, Y 0.8569, Z -3.8333, A 0.000, B 0.000, C 0.000 }
gfCNCPoint3[2378] = {X -0.0965, Y 8.7891, Z -3.8333, A 0.000, B 0.000, C 0.000 }
gfCNCPoint3[2379] = {X -0.7633, Y 8.9979, Z -3.8333, A 0.000, B 0.000, C 0.000 }
gfCNCPoint3[2380] = {X -1.3934, Y 9.2998, Z -3.8333, A 0.000, B 0.000, C 0.000 }
gfCNCPoint3[2381] = {X -1.9904, Y 9.6404, Z -3.8333, A 0.000, B 0.000, C 0.000 }
gfCNCPoint3[2382] = {X -2.6455, Y 10.0884, Z -3.8333, A 0.000, B 0.000, C 0.000 }
gfCNCPoint3[2383] = {X -3.2192, Y 10.6366, Z -3.8333, A 0.000, B 0.000, C 0.000 }
gfCNCPoint3[2384] = {X -3.6965, Y 11.2706, Z -3.8333, A 0.000, B 0.000, C 0.000 }
gfCNCPoint3[2385] = {X -3.6965, Y 12.3462, Z -3.8333, A 0.000, B 0.000, C 0.000 }
gfCNCPoint3[2386] = {X -3.2332, Y 11.4384, Z -3.8333, A 0.000, B 0.000, C 0.000 }
gfCNCPoint3[2387] = {X -2.5734, Y 10.6615, Z -3.8333, A 0.000, B 0.000, C 0.000 }
gfCNCPoint3[2388] = {X -1.7526, Y 10.0573, Z -3.8333, A 0.000, B 0.000, C 0.000 }
gfCNCPoint3[2389] = {X -1.0994, Y 9.6852, Z -3.8333, A 0.000, B 0.000, C 0.000 }
gfCNCPoint3[2390] = {X -0.1608, Y 9.3012, Z -3.8333, A 0.000, B 0.000, C 0.000 }
gfCNCPoint3[2391] = {X 0.8408, Y 9.1423, Z -3.8333, A 0.000, B 0.000, C 0.000 }
gfCNCPoint3[2392] = {X 1.8522, Y 9.2169, Z -3.8333, A 0.000, B 0.000, C 0.000 }
gfCNCPoint3[2393] = {X 2.2357, Y 9.3083, Z -3.8333, A 0.000, B 0.000, C 0.000 }
gfCNCPoint3[2394] = {X 2.6096, Y 9.4337, Z -3.8333, A 0.000, B 0.000, C 0.000 }
gfCNCPoint3[2395] = {X 3.3780, Y 9.0736, Z -3.8333, A 0.000, B 0.000, C 0.000 }
gfCNCPoint3[2396] = {X 4.1699, Y 8.7685, Z -3.8333, A 0.000, B 0.000, C 0.000 }
gfCNCPoint3[2397] = {X 6.0871, Y 8.0978, Z -3.8333, A 0.000, B 0.000, C 0.000 }
gfCNCPoint3[2398] = {X 8.0549, Y 7.5949, Z -3.8333, A 0.000, B 0.000, C 0.000 }
gfCNCPoint3[2399] = {X 10.0588, Y 7.2635, Z -3.8333, A 0.000, B 0.000, C 0.000 }
gfCNCPoint3[2400] = {X 12.0838, Y 7.1061, Z -3.8333, A 0.000, B 0.000, C 0.000 }
gfCNCPoint3[2401] = {X 14.1148, Y 7.1239, Z -3.8333, A 0.000, B 0.000, C 0.000 }
gfCNCPoint3[2402] = {X 16.1367, Y 7.3167, Z -3.8333, A 0.000, B 0.000, C 0.000 }
gfCNCPoint3[2403] = {X 16.5418, Y 7.3732, Z -3.8333, A 0.000, B 0.000, C 0.000 }
gfCNCPoint3[2404] = {X 18.2857, Y 7.7306, Z -3.8333, A 0.000, B 0.000, C 0.000 }
gfCNCPoint3[2405] = {X 19.9845, Y 8.2629, Z -3.8333, A 0.000, B 0.000, C 0.000 }
gfCNCPoint3[2406] = {X 21.6204, Y 8.9648, Z -3.8333, A 0.000, B 0.000, C 0.000 }
gfCNCPoint3[2407] = {X 23.1768, Y 9.8289, Z -3.8333, A 0.000, B 0.000, C 0.000 }
gfCNCPoint3[2408] = {X 24.6376, Y 10.8464, Z -3.8333, A 0.000, B 0.000, C 0.000 }
gfCNCPoint3[2409] = {X 25.7300, Y 11.8017, Z -3.8333, A 0.000, B 0.000, C 0.000 }
gfCNCPoint3[2410] = {X 26.7098, Y 12.8722, Z -3.8333, A 0.000, B 0.000, C 0.000 }
gfCNCPoint3[2411] = {X 27.5649, Y 14.0447, Z -3.8333, A 0.000, B 0.000, C 0.000 }
gfCNCPoint3[2412] = {X 28.2849, Y 15.3047, Z -3.8333, A 0.000, B 0.000, C 0.000 }
gfCNCPoint3[2413] = {X 28.8608, Y 16.6368, Z -3.8333, A 0.000, B 0.000, C 0.000 }
gfCNCPoint3[2414] = {X 29.3372, Y 18.3013, Z -3.8333, A 0.000, B 0.000, C 0.000 }
gfCNCPoint3[2415] = {X 29.6198, Y 20.0095, Z -3.8333, A 0.000, B 0.000, C 0.000 }
gfCNCPoint3[2416] = {X 29.7050, Y 21.7387, Z -3.8333, A 0.000, B 0.000, C 0.000 }
gfCNCPoint3[2417] = {X 29.5916, Y 23.4664, Z -3.8333, A 0.000, B 0.000, C 0.000 }
gfCNCPoint3[2418] = {X 29.2811, Y 25.1696, Z -3.8333, A 0.000, B 0.000, C 0.000 }
gfCNCPoint3[2419] = {X 28.9105, Y 26.4228, Z -3.8333, A 0.000, B 0.000, C 0.000 }
gfCNCPoint3[2420] = {X 28.4032, Y 27.6272, Z -3.8333, A 0.000, B 0.000, C 0.000 }
gfCNCPoint3[2421] = {X 27.7655, Y 28.7679, Z -3.8333, A 0.000, B 0.000, C 0.000 }
gfCNCPoint3[2422] = {X 27.4793, Y 29.1979, Z -3.8333, A 0.000, B 0.000, C 0.000 }
gfCNCPoint3[2423] = {X 27.1745, Y 29.6149, Z -3.8333, A 0.000, B 0.000, C 0.000 }
gfCNCPoint3[2424] = {X 26.5418, Y 30.3736, Z -3.8333, A 0.000, B 0.000, C 0.000 }
gfCNCPoint3[2425] = {X 25.8477, Y 31.0766, Z -3.8333, A 0.000, B 0.000, C 0.000 }
gfCNCPoint3[2426] = {X 25.6474, Y 31.2589, Z -3.8333, A 0.000, B 0.000, C 0.000 }
gfCNCPoint3[2427] = {X 25.4428, Y 31.4366, Z -3.8333, A 0.000, B 0.000, C 0.000 }
gfCNCPoint3[2428] = {X 25.6934, Y 31.5322, Z -3.8333, A 0.000, B 0.000, C 0.000 }
gfCNCPoint3[2429] = {X 25.9378, Y 31.6429, Z -3.8333, A 0.000, B 0.000, C 0.000 }
gfCNCPoint3[2430] = {X 26.6625, Y 32.0901, Z -3.8333, A 0.000, B 0.000, C 0.000 }
